SPLINE
SPL {X  -162.820, Y  +465.690, Z    +0.000, E1   -36.140, E3 +383343.973}
SPL {X  -162.820, Y  +470.432, Z    +0.000, E1   -36.100, E3 +383357.855}
SPL {X  -162.820, Y  +475.701, Z    +0.000, E1   -36.157, E3 +383372.483}
SPL {X  -162.820, Y  +479.954, Z    +0.000, E1   -36.086, E3 +383385.023}
SPL {X  -162.820, Y  +485.438, Z    +0.000, E1   -36.112, E3 +383400.741}
SPL {X  -162.820, Y  +490.843, Z    +0.000, E1   -36.087, E3 +383416.154}
SPL {X  -162.820, Y  +494.712, Z    +0.000, E1   -36.164, E3 +383426.667}
SPL {X  -162.820, Y  +497.796, Z    +0.000, E1   -36.022, E3 +383436.373}
SPL {X  -162.820, Y  +502.146, Z    +0.000, E1   -36.123, E3 +383448.242}
SPL {X  -162.820, Y  +505.688, Z    +0.000, E1   -36.050, E3 +383458.724}
SPL {X  -162.820, Y  +509.364, Z    +0.000, E1   -36.084, E3 +383469.095}
SPL {X  -162.820, Y  +513.393, Z    +0.000, E1   -36.179, E3 +383479.950}
SPL {X  -162.820, Y  +516.436, Z    +0.000, E1   -36.094, E3 +383489.146}
SPL {X  -162.820, Y  +520.482, Z    +0.000, E1   -36.096, E3 +383500.778}
SPL {X  -162.820, Y  +524.107, Z    +0.000, E1   -36.045, E3 +383511.362}
SPL {X  -162.820, Y  +527.962, Z    +0.000, E1   -36.074, E3 +383522.295}
SPL {X  -162.820, Y  +532.253, Z    +0.000, E1   -36.170, E3 +383533.884}
SPL {X  -162.820, Y  +536.031, Z    +0.000, E1   -36.058, E3 +383545.422}
SPL {X  -162.820, Y  +541.179, Z    +0.000, E1   -36.085, E3 +383560.062}
SPL {X  -162.820, Y  +546.355, Z    +0.000, E1   -36.114, E3 +383574.607}
SPL {X  -162.820, Y  +551.776, Z    +0.000, E1   -36.108, E3 +383590.240}
SPL {X  -162.820, Y  +558.272, Z    +0.000, E1   -36.170, E3 +383608.449}
SPL {X  -162.820, Y  +562.721, Z    +0.000, E1   -36.046, E3 +383621.674}
SPL {X  -162.820, Y  +566.500, Z    +0.000, E1   -36.073, E3 +383632.406}
SPL {X  -162.820, Y  +570.319, Z    +0.000, E1   -36.045, E3 +383643.434}
SPL {X  -162.820, Y  +573.265, Z    +0.000, E1   -36.071, E3 +383651.671}
SPL {X  -162.820, Y  +576.887, Z    +0.000, E1   -36.084, E3 +383662.029}
SPL {X  -162.820, Y  +581.763, Z    +0.000, E1   -36.093, E3 +383675.966}
SPL {X  -162.820, Y  +586.693, Z    +0.000, E1   -36.086, E3 +383690.071}
SPL {X  -162.820, Y  +591.665, Z    +0.000, E1   -36.045, E3 +383704.599}
SPL {X  -162.820, Y  +597.399, Z    +0.000, E1   -36.147, E3 +383720.362}
SPL {X  -162.820, Y  +602.243, Z    +0.000, E1   -36.085, E3 +383734.508}
SPL {X  -162.820, Y  +605.848, Z    +0.000, E1   -36.070, E3 +383744.829}
SPL {X  -162.820, Y  +609.375, Z    +0.000, E1   -36.084, E3 +383754.879}
SPL {X  -162.820, Y  +612.959, Z    +0.000, E1   -36.034, E3 +383765.400}
SPL {X  -162.820, Y  +616.897, Z    +0.000, E1   -36.061, E3 +383776.547}
SPL {X  -162.820, Y  +621.516, Z    +0.000, E1   -36.072, E3 +383789.746}
SPL {X  -162.820, Y  +626.243, Z    +0.000, E1   -36.105, E3 +383802.989}
SPL {X  -162.820, Y  +630.571, Z    +0.000, E1   -36.057, E3 +383815.691}
SPL {X  -162.820, Y  +634.189, Z    +0.000, E1   -36.065, E3 +383825.885}
SPL {X  -162.820, Y  +638.473, Z    +0.000, E1   -36.098, E3 +383838.122}
SPL {X  -162.820, Y  +642.832, Z    +0.000, E1   -36.091, E3 +383850.448}
SPL {X  -162.820, Y  +646.320, Z    +0.000, E1   -36.078, E3 +383860.555}
SPL {X  -162.820, Y  +649.997, Z    +0.000, E1   -36.000, E3 +383871.525}
SPL {X  -162.820, Y  +655.571, Z    +0.000, E1   -36.141, E3 +383886.860}
SPL {X  -162.820, Y  +661.560, Z    +0.000, E1   -36.068, E3 +383904.287}
SPL {X  -162.820, Y  +667.641, Z    +0.000, E1   -36.092, E3 +383921.668}
SPL {X  -162.820, Y  +673.415, Z    +0.000, E1   -36.053, E3 +383938.259}
SPL {X  -162.761, Y  +677.889, Z    +0.000, E1   -36.122, E3 +383950.577}
SPL {X  -162.577, Y  +682.401, Z    +0.000, E1   -36.021, E3 +383964.193}
SPL {X  -162.187, Y  +687.846, Z    +0.000, E1   -36.007, E3 +383979.862}
SPL {X  -161.667, Y  +692.839, Z    +0.000, E1   -35.918, E3 +383994.628}
SPL {X  -161.078, Y  +697.256, Z    +0.000, E1   -35.797, E3 +384007.964}
SPL {X  -160.313, Y  +701.964, Z    +0.000, E1   -35.709, E3 +384022.039}
SPL {X  -159.317, Y  +707.091, Z    +0.000, E1   -35.482, E3 +384038.063}
SPL {X  -158.510, Y  +710.714, Z    +0.000, E1   -35.230, E3 +384049.774}
SPL {X  -155.037, Y  +723.239, Z    +0.000, E1   -39.382, E3 +384058.870}
SPL {X  -152.141, Y  +731.494, Z    +0.000, E1   -35.181, E3 +384117.676}
ENDSPLINE

SPLINE
SPL {X  -152.670, Y  +730.088, Z    +0.000, E1   -30.916, E3 +384191.038}
SPL {X  -160.727, Y  +699.521, Z    +0.000, E1   -18.202, E3 +384157.321}
SPL {X  -161.979, Y  +690.023, Z    +0.000, E1   -12.991, E3 +384164.131}
SPL {X  -162.641, Y  +681.139, Z    +0.000, E1    -7.893, E3 +384166.223}
SPL {X  -162.820, Y  +673.062, Z    +0.000, E1    -2.992, E3 +384165.190}
SPL {X  -162.820, Y  +666.731, Z    +0.000, E1    +1.545, E3 +384166.820}
SPL {X  -162.820, Y  +660.758, Z    +0.000, E1    +6.523, E3 +384166.530}
SPL {X  -162.820, Y  +650.583, Z    +0.000, E1   +16.035, E3 +384165.503}
SPL {X  -162.820, Y  +629.267, Z    +0.000, E1   +31.872, E3 +384176.651}
SPL {X  -162.820, Y  +620.680, Z    +0.000, E1   +34.107, E3 +384190.701}
SPL {X  -162.820, Y  +601.185, Z    +0.000, E1   +39.430, E3 +384214.208}
SPL {X  -162.820, Y  +599.927, Z    +0.000, E1   +35.241, E3 +384240.786}
SPL {X  -162.820, Y  +599.021, Z    +0.000, E1   +33.912, E3 +384251.837}
SPL {X  -162.820, Y  +595.170, Z    +0.000, E1   +33.784, E3 +384264.743}
SPL {X  -162.820, Y  +589.785, Z    +0.000, E1   +33.904, E3 +384280.740}
SPL {X  -162.820, Y  +584.646, Z    +0.000, E1   +33.882, E3 +384296.809}
SPL {X  -162.820, Y  +579.919, Z    +0.000, E1   +33.857, E3 +384311.597}
SPL {X  -162.820, Y  +574.615, Z    +0.000, E1   +33.920, E3 +384327.771}
SPL {X  -162.820, Y  +569.298, Z    +0.000, E1   +33.851, E3 +384344.633}
SPL {X  -162.820, Y  +563.983, Z    +0.000, E1   +33.916, E3 +384360.774}
SPL {X  -162.820, Y  +559.395, Z    +0.000, E1   +33.796, E3 +384375.655}
SPL {X  -162.820, Y  +554.453, Z    +0.000, E1   +33.841, E3 +384390.880}
SPL {X  -162.820, Y  +548.576, Z    +0.000, E1   +33.950, E3 +384408.410}
SPL {X  -162.820, Y  +544.808, Z    +0.000, E1   +33.827, E3 +384420.673}
SPL {X  -162.820, Y  +541.668, Z    +0.000, E1   +33.787, E3 +384430.779}
SPL {X  -162.820, Y  +537.061, Z    +0.000, E1   +33.897, E3 +384444.437}
SPL {X  -162.820, Y  +532.164, Z    +0.000, E1   +33.861, E3 +384459.911}
SPL {X  -162.820, Y  +526.783, Z    +0.000, E1   +33.870, E3 +384476.594}
SPL {X  -162.820, Y  +521.520, Z    +0.000, E1   +33.826, E3 +384493.241}
SPL {X  -162.820, Y  +515.754, Z    +0.000, E1   +33.911, E3 +384510.643}
SPL {X  -162.820, Y  +510.207, Z    +0.000, E1   +33.879, E3 +384528.023}
SPL {X  -162.820, Y  +505.651, Z    +0.000, E1   +33.839, E3 +384542.317}
SPL {X  -162.820, Y  +500.931, Z    +0.000, E1   +34.256, E3 +384554.190}
SPL {X  -162.820, Y  +481.122, Z    +0.000, E1   +41.279, E3 +384564.455}
SPL {X  -162.820, Y  +478.698, Z    +0.000, E1   +40.526, E3 +384574.804}
SPL {X  -162.820, Y  +475.203, Z    +0.000, E1   +39.596, E3 +384589.263}
SPL {X  -162.820, Y  +472.097, Z    +0.000, E1   +38.411, E3 +384604.230}
SPL {X  -162.820, Y  +469.308, Z    +0.000, E1   +37.839, E3 +384615.034}
SPL {X  -162.820, Y  +467.216, Z    +0.000, E1   +37.215, E3 +384624.601}
SPL {X  -162.820, Y  +462.598, Z    +0.000, E1   +37.325, E3 +384636.555}
SPL {X  -162.820, Y  +457.832, Z    +0.000, E1   +37.294, E3 +384649.841}
SPL {X  -162.820, Y  +452.986, Z    +0.000, E1   +37.368, E3 +384662.575}
SPL {X  -162.820, Y  +447.084, Z    +0.000, E1   +37.389, E3 +384678.766}
SPL {X  -162.820, Y  +440.036, Z    +0.000, E1   +37.326, E3 +384698.384}
SPL {X  -162.820, Y  +434.320, Z    +0.000, E1   +37.343, E3 +384713.707}
SPL {X  -162.820, Y  +430.091, Z    +0.000, E1   +37.424, E3 +384724.707}
SPL {X  -162.820, Y  +426.177, Z    +0.000, E1   +37.250, E3 +384736.530}
SPL {X  -162.820, Y  +421.391, Z    +0.000, E1   +37.346, E3 +384748.994}
SPL {X  -162.820, Y  +416.811, Z    +0.000, E1   +37.348, E3 +384761.528}
SPL {X  -162.820, Y  +411.860, Z    +0.000, E1   +37.402, E3 +384774.680}
SPL {X  -162.820, Y  +407.726, Z    +0.000, E1   +37.291, E3 +384786.627}
SPL {X  -162.820, Y  +403.543, Z    +0.000, E1   +37.305, E3 +384797.973}
SPL {X  -162.820, Y  +399.300, Z    +0.000, E1   +37.355, E3 +384809.257}
SPL {X  -162.820, Y  +395.182, Z    +0.000, E1   +37.347, E3 +384820.546}
SPL {X  -162.820, Y  +390.797, Z    +0.000, E1   +37.358, E3 +384832.458}
SPL {X  -162.820, Y  +386.671, Z    +0.000, E1   +37.363, E3 +384843.639}
SPL {X  -162.820, Y  +382.174, Z    +0.000, E1   +37.329, E3 +384856.217}
SPL {X  -162.785, Y  +377.133, Z    +0.000, E1   +37.299, E3 +384870.146}
SPL {X  -162.623, Y  +372.484, Z    +0.000, E1   +37.337, E3 +384882.586}
SPL {X  -162.331, Y  +367.894, Z    +0.000, E1   +37.251, E3 +384895.698}
SPL {X  -161.920, Y  +363.407, Z    +0.000, E1   +37.164, E3 +384908.432}
SPL {X  -161.482, Y  +359.669, Z    +0.000, E1   +37.064, E3 +384919.217}
SPL {X  -160.943, Y  +355.851, Z    +0.000, E1   +37.136, E3 +384929.203}
SPL {X  -160.493, Y  +353.069, Z    +0.000, E1   +36.789, E3 +384938.855}
SPL {X  -159.837, Y  +349.474, Z    +0.000, E1   +36.824, E3 +384948.521}
SPL {X  -158.862, Y  +344.820, Z    +0.000, E1   +36.732, E3 +384961.884}
SPL {X  -157.959, Y  +341.011, Z    +0.000, E1   +36.448, E3 +384973.780}
SPL {X  -153.520, Y  +326.260, Z    +0.000, E1   +41.363, E3 +384982.613}
SPL {X  -150.942, Y  +319.452, Z    +0.000, E1   +36.529, E3 +385038.970}
ENDSPLINE

SPLINE
SPL {X  -159.264, Y  +346.659, Z    +0.000, E1   +22.083, E3 +385079.544}
SPL {X  -161.245, Y  +357.907, Z    +0.000, E1   +16.095, E3 +385092.977}
SPL {X  -162.697, Y  +374.161, Z    +0.000, E1    +7.119, E3 +385090.966}
SPL {X  -162.820, Y  +380.878, Z    +0.000, E1    +2.854, E3 +385093.797}
SPL {X  -162.820, Y  +385.313, Z    +0.000, E1    -0.228, E3 +385093.578}
SPL {X  -162.820, Y  +389.965, Z    +0.000, E1    -3.918, E3 +385092.946}
SPL {X  -162.820, Y  +394.532, Z    +0.000, E1    -7.849, E3 +385094.494}
SPL {X  -162.820, Y  +400.765, Z    +0.000, E1   -14.108, E3 +385091.961}
SPL {X  -162.820, Y  +411.829, Z    +0.000, E1   -24.195, E3 +385094.039}
SPL {X  -162.820, Y  +434.900, Z    +0.000, E1   -34.666, E3 +385121.403}
SPL {X  -162.820, Y  +465.031, Z    +0.000, E1   -41.710, E3 +385159.076}
SPL {X  -162.820, Y  +465.893, Z    +0.000, E1   -40.572, E3 +385167.605}
ENDSPLINE

SPLINE
SPL {X  -162.820, Y  +458.794, Z    +0.000, E1   -36.100, E3 +385176.334}
ENDSPLINE

SPLINE
SPL {X  -162.820, Y  +461.779, Z    +0.000, E1   -35.988, E3 +385185.530}
SPL {X  -162.820, Y  +465.690, Z    +0.000, E1   -36.140, E3 +385195.825}
SPL {X  -162.820, Y  +470.432, Z    +0.000, E1   -36.100, E3 +385209.707}
SPL {X  -162.820, Y  +475.701, Z    +0.000, E1   -36.157, E3 +385224.334}
SPL {X  -162.820, Y  +479.954, Z    +0.000, E1   -36.086, E3 +385236.875}
SPL {X  -162.820, Y  +483.976, Z    +0.000, E1   -36.049, E3 +385248.607}
SPL {X  -162.820, Y  +488.601, Z    +0.000, E1   -36.081, E3 +385261.697}
SPL {X  -162.820, Y  +493.837, Z    +0.000, E1   -36.178, E3 +385276.040}
SPL {X  -162.820, Y  +498.932, Z    +0.000, E1   -36.079, E3 +385291.245}
SPL {X  -162.820, Y  +504.528, Z    +0.000, E1   -36.109, E3 +385307.041}
SPL {X  -162.820, Y  +509.364, Z    +0.000, E1   -36.084, E3 +385320.946}
SPL {X  -162.820, Y  +515.001, Z    +0.000, E1   -36.183, E3 +385336.584}
SPL {X  -162.820, Y  +520.482, Z    +0.000, E1   -36.096, E3 +385352.630}
SPL {X  -162.820, Y  +524.107, Z    +0.000, E1   -36.045, E3 +385363.214}
SPL {X  -162.820, Y  +527.962, Z    +0.000, E1   -36.074, E3 +385374.146}
SPL {X  -162.820, Y  +532.253, Z    +0.000, E1   -36.170, E3 +385385.735}
SPL {X  -162.820, Y  +536.031, Z    +0.000, E1   -36.058, E3 +385397.273}
SPL {X  -162.820, Y  +541.179, Z    +0.000, E1   -36.085, E3 +385411.914}
SPL {X  -162.820, Y  +546.355, Z    +0.000, E1   -36.114, E3 +385426.458}
SPL {X  -162.820, Y  +551.776, Z    +0.000, E1   -36.108, E3 +385442.092}
SPL {X  -162.820, Y  +556.944, Z    +0.000, E1   -36.118, E3 +385456.663}
SPL {X  -162.820, Y  +561.684, Z    +0.000, E1   -36.118, E3 +385470.255}
SPL {X  -162.820, Y  +566.500, Z    +0.000, E1   -36.073, E3 +385484.258}
SPL {X  -162.820, Y  +571.734, Z    +0.000, E1   -36.094, E3 +385499.187}
SPL {X  -162.820, Y  +576.887, Z    +0.000, E1   -36.084, E3 +385513.881}
SPL {X  -162.820, Y  +581.763, Z    +0.000, E1   -36.093, E3 +385527.818}
SPL {X  -162.820, Y  +586.693, Z    +0.000, E1   -36.086, E3 +385541.923}
SPL {X  -162.820, Y  +591.665, Z    +0.000, E1   -36.045, E3 +385556.450}
SPL {X  -162.820, Y  +597.399, Z    +0.000, E1   -36.147, E3 +385572.214}
SPL {X  -162.820, Y  +602.243, Z    +0.000, E1   -36.085, E3 +385586.360}
SPL {X  -162.820, Y  +606.975, Z    +0.000, E1   -36.102, E3 +385599.805}
SPL {X  -162.820, Y  +611.980, Z    +0.000, E1   -36.072, E3 +385614.351}
SPL {X  -162.820, Y  +616.897, Z    +0.000, E1   -36.061, E3 +385628.399}
SPL {X  -162.820, Y  +621.516, Z    +0.000, E1   -36.072, E3 +385641.598}
SPL {X  -162.820, Y  +626.243, Z    +0.000, E1   -36.105, E3 +385654.841}
SPL {X  -162.820, Y  +630.571, Z    +0.000, E1   -36.057, E3 +385667.543}
SPL {X  -162.820, Y  +635.505, Z    +0.000, E1   -36.079, E3 +385681.549}
SPL {X  -162.820, Y  +641.277, Z    +0.000, E1   -36.126, E3 +385697.841}
SPL {X  -162.820, Y  +646.320, Z    +0.000, E1   -36.078, E3 +385712.407}
SPL {X  -162.820, Y  +651.289, Z    +0.000, E1   -36.059, E3 +385726.863}
SPL {X  -162.820, Y  +656.677, Z    +0.000, E1   -36.110, E3 +385741.876}
SPL {X  -162.820, Y  +661.560, Z    +0.000, E1   -36.068, E3 +385756.139}
SPL {X  -162.820, Y  +667.641, Z    +0.000, E1   -36.092, E3 +385773.520}
SPL {X  -162.820, Y  +673.415, Z    +0.000, E1   -36.053, E3 +385790.111}
SPL {X  -162.761, Y  +677.889, Z    +0.000, E1   -36.122, E3 +385802.429}
SPL {X  -162.577, Y  +682.401, Z    +0.000, E1   -36.021, E3 +385816.045}
SPL {X  -162.296, Y  +686.558, Z    +0.000, E1   -35.952, E3 +385828.236}
SPL {X  -161.948, Y  +690.331, Z    +0.000, E1   -35.960, E3 +385839.034}
SPL {X  -161.544, Y  +693.846, Z    +0.000, E1   -35.908, E3 +385849.309}
SPL {X  -160.925, Y  +698.267, Z    +0.000, E1   -35.816, E3 +385862.741}
SPL {X  -160.151, Y  +702.861, Z    +0.000, E1   -35.643, E3 +385876.711}
SPL {X  -159.317, Y  +707.091, Z    +0.000, E1   -35.482, E3 +385889.915}
SPL {X  -158.510, Y  +710.714, Z    +0.000, E1   -35.230, E3 +385901.626}
SPL {X  -155.037, Y  +723.239, Z    +0.000, E1   -39.382, E3 +385910.722}
SPL {X  -152.141, Y  +731.494, Z    +0.000, E1   -35.181, E3 +385969.528}
ENDSPLINE

SPLINE
SPL {X  -152.670, Y  +730.088, Z    +0.000, E1   -30.916, E3 +386042.890}
SPL {X  -160.727, Y  +699.521, Z    +0.000, E1   -18.202, E3 +386009.173}
SPL {X  -161.979, Y  +690.023, Z    +0.000, E1   -12.991, E3 +386015.983}
SPL {X  -162.641, Y  +681.139, Z    +0.000, E1    -7.893, E3 +386018.075}
SPL {X  -162.815, Y  +674.833, Z    +0.000, E1    -4.093, E3 +386015.690}
SPL {X  -162.820, Y  +669.862, Z    +0.000, E1    -0.751, E3 +386018.909}
SPL {X  -162.820, Y  +664.572, Z    +0.000, E1    +3.252, E3 +386018.722}
SPL {X  -162.820, Y  +657.781, Z    +0.000, E1    +9.391, E3 +386016.545}
SPL {X  -162.820, Y  +648.706, Z    +0.000, E1   +17.761, E3 +386018.297}
SPL {X  -162.820, Y  +635.926, Z    +0.000, E1   +28.192, E3 +386023.124}
SPL {X  -162.820, Y  +621.673, Z    +0.000, E1   +34.265, E3 +386039.482}
SPL {X  -162.820, Y  +609.002, Z    +0.000, E1   +38.458, E3 +386052.704}
SPL {X  -162.820, Y  +596.392, Z    +0.000, E1   +37.895, E3 +386086.173}
ENDSPLINE

SPLINE
SPL {X  -162.820, Y  +601.432, Z    +0.000, E1   +34.026, E3 +386095.470}
ENDSPLINE

SPLINE
SPL {X  -162.820, Y  +597.570, Z    +0.000, E1   +33.919, E3 +386108.368}
SPL {X  -162.820, Y  +592.692, Z    +0.000, E1   +33.779, E3 +386124.260}
SPL {X  -162.820, Y  +588.795, Z    +0.000, E1   +33.876, E3 +386135.697}
SPL {X  -162.820, Y  +584.646, Z    +0.000, E1   +33.882, E3 +386148.661}
SPL {X  -162.820, Y  +579.919, Z    +0.000, E1   +33.857, E3 +386163.449}
SPL {X  -162.820, Y  +576.636, Z    +0.000, E1   +33.845, E3 +386173.595}
SPL {X  -162.820, Y  +573.566, Z    +0.000, E1   +33.899, E3 +386182.844}
SPL {X  -162.820, Y  +570.335, Z    +0.000, E1   +33.821, E3 +386193.328}
SPL {X  -162.820, Y  +565.901, Z    +0.000, E1   +33.889, E3 +386206.849}
SPL {X  -162.820, Y  +562.173, Z    +0.000, E1   +33.897, E3 +386218.140}
SPL {X  -162.820, Y  +558.179, Z    +0.000, E1   +33.857, E3 +386231.075}
SPL {X  -162.820, Y  +553.486, Z    +0.000, E1   +33.777, E3 +386245.980}
SPL {X  -162.820, Y  +549.726, Z    +0.000, E1   +33.905, E3 +386256.835}
SPL {X  -162.820, Y  +545.760, Z    +0.000, E1   +33.901, E3 +386269.231}
SPL {X  -162.820, Y  +541.668, Z    +0.000, E1   +33.787, E3 +386282.631}
SPL {X  -162.820, Y  +538.174, Z    +0.000, E1   +33.865, E3 +386292.920}
SPL {X  -162.820, Y  +534.943, Z    +0.000, E1   +33.919, E3 +386302.661}
SPL {X  -162.820, Y  +531.459, Z    +0.000, E1   +33.783, E3 +386314.318}
SPL {X  -162.820, Y  +526.783, Z    +0.000, E1   +33.870, E3 +386328.446}
SPL {X  -162.820, Y  +521.520, Z    +0.000, E1   +33.826, E3 +386345.093}
SPL {X  -162.820, Y  +516.814, Z    +0.000, E1   +33.917, E3 +386358.994}
SPL {X  -162.820, Y  +512.685, Z    +0.000, E1   +33.830, E3 +386372.437}
SPL {X  -162.820, Y  +508.888, Z    +0.000, E1   +33.871, E3 +386383.852}
SPL {X  -162.820, Y  +505.651, Z    +0.000, E1   +33.839, E3 +386394.169}
SPL {X  -162.820, Y  +500.931, Z    +0.000, E1   +34.256, E3 +386406.042}
SPL {X  -162.820, Y  +481.122, Z    +0.000, E1   +41.279, E3 +386416.307}
SPL {X  -162.820, Y  +478.698, Z    +0.000, E1   +40.526, E3 +386426.656}
SPL {X  -162.820, Y  +475.203, Z    +0.000, E1   +39.596, E3 +386441.115}
SPL {X  -162.820, Y  +472.097, Z    +0.000, E1   +38.411, E3 +386456.082}
SPL {X  -162.820, Y  +469.308, Z    +0.000, E1   +37.839, E3 +386466.886}
SPL {X  -162.820, Y  +467.216, Z    +0.000, E1   +37.215, E3 +386476.452}
SPL {X  -162.820, Y  +462.598, Z    +0.000, E1   +37.325, E3 +386488.407}
SPL {X  -162.820, Y  +459.177, Z    +0.000, E1   +37.207, E3 +386498.434}
SPL {X  -162.820, Y  +453.939, Z    +0.000, E1   +37.397, E3 +386511.786}
SPL {X  -162.820, Y  +447.084, Z    +0.000, E1   +37.389, E3 +386530.618}
SPL {X  -162.820, Y  +440.036, Z    +0.000, E1   +37.326, E3 +386550.235}
SPL {X  -162.820, Y  +434.320, Z    +0.000, E1   +37.343, E3 +386565.559}
SPL {X  -162.820, Y  +430.091, Z    +0.000, E1   +37.424, E3 +386576.559}
SPL {X  -162.820, Y  +426.177, Z    +0.000, E1   +37.250, E3 +386588.382}
SPL {X  -162.820, Y  +421.391, Z    +0.000, E1   +37.346, E3 +386600.845}
SPL {X  -162.820, Y  +416.811, Z    +0.000, E1   +37.348, E3 +386613.380}
SPL {X  -162.820, Y  +411.860, Z    +0.000, E1   +37.402, E3 +386626.531}
SPL {X  -162.820, Y  +407.726, Z    +0.000, E1   +37.291, E3 +386638.479}
SPL {X  -162.820, Y  +403.543, Z    +0.000, E1   +37.305, E3 +386649.825}
SPL {X  -162.820, Y  +399.300, Z    +0.000, E1   +37.355, E3 +386661.109}
SPL {X  -162.820, Y  +395.182, Z    +0.000, E1   +37.347, E3 +386672.398}
SPL {X  -162.820, Y  +390.797, Z    +0.000, E1   +37.358, E3 +386684.310}
SPL {X  -162.820, Y  +386.671, Z    +0.000, E1   +37.363, E3 +386695.491}
SPL {X  -162.820, Y  +382.174, Z    +0.000, E1   +37.329, E3 +386708.069}
SPL {X  -162.785, Y  +377.133, Z    +0.000, E1   +37.299, E3 +386721.998}
SPL {X  -162.576, Y  +371.586, Z    +0.000, E1   +37.322, E3 +386737.110}
SPL {X  -162.256, Y  +366.963, Z    +0.000, E1   +37.251, E3 +386749.999}
SPL {X  -161.920, Y  +363.407, Z    +0.000, E1   +37.164, E3 +386760.284}
SPL {X  -161.341, Y  +358.603, Z    +0.000, E1   +37.117, E3 +386773.764}
SPL {X  -160.616, Y  +353.801, Z    +0.000, E1   +36.942, E3 +386787.929}
SPL {X  -159.837, Y  +349.474, Z    +0.000, E1   +36.824, E3 +386800.373}
SPL {X  -158.862, Y  +344.820, Z    +0.000, E1   +36.732, E3 +386813.735}
SPL {X  -157.959, Y  +341.011, Z    +0.000, E1   +36.448, E3 +386825.632}
SPL {X  -153.520, Y  +326.260, Z    +0.000, E1   +41.363, E3 +386834.465}
SPL {X  -150.942, Y  +319.452, Z    +0.000, E1   +36.529, E3 +386890.821}
ENDSPLINE

SPLINE
SPL {X  -159.264, Y  +346.659, Z    +0.000, E1   +22.083, E3 +386931.396}
SPL {X  -161.245, Y  +357.907, Z    +0.000, E1   +16.095, E3 +386944.828}
SPL {X  -162.697, Y  +374.161, Z    +0.000, E1    +7.119, E3 +386942.818}
SPL {X  -162.820, Y  +380.878, Z    +0.000, E1    +2.854, E3 +386945.649}
SPL {X  -162.820, Y  +385.313, Z    +0.000, E1    -0.228, E3 +386945.429}
SPL {X  -162.820, Y  +389.965, Z    +0.000, E1    -3.918, E3 +386944.798}
SPL {X  -162.820, Y  +394.532, Z    +0.000, E1    -7.849, E3 +386946.346}
SPL {X  -162.820, Y  +400.765, Z    +0.000, E1   -14.108, E3 +386943.813}
SPL {X  -162.820, Y  +411.829, Z    +0.000, E1   -24.195, E3 +386945.890}
SPL {X  -162.820, Y  +434.900, Z    +0.000, E1   -34.666, E3 +386973.255}
SPL {X  -162.820, Y  +465.440, Z    +0.000, E1   -41.264, E3 +387014.562}
ENDSPLINE

SPLINE
SPL {X  -162.820, Y  +458.794, Z    +0.000, E1   -36.100, E3 +387028.186}
ENDSPLINE

SPLINE
SPL {X  -162.820, Y  +461.779, Z    +0.000, E1   -35.988, E3 +387037.382}
SPL {X  -162.820, Y  +465.690, Z    +0.000, E1   -36.140, E3 +387047.676}
SPL {X  -162.820, Y  +470.432, Z    +0.000, E1   -36.100, E3 +387061.559}
SPL {X  -162.820, Y  +475.701, Z    +0.000, E1   -36.157, E3 +387076.186}
SPL {X  -162.820, Y  +479.954, Z    +0.000, E1   -36.086, E3 +387088.727}
SPL {X  -162.820, Y  +483.976, Z    +0.000, E1   -36.049, E3 +387100.459}
SPL {X  -162.820, Y  +489.628, Z    +0.000, E1   -36.135, E3 +387116.289}
SPL {X  -162.820, Y  +494.712, Z    +0.000, E1   -36.164, E3 +387130.370}
SPL {X  -162.820, Y  +498.932, Z    +0.000, E1   -36.079, E3 +387143.097}
SPL {X  -162.820, Y  +504.528, Z    +0.000, E1   -36.109, E3 +387158.893}
SPL {X  -162.820, Y  +509.364, Z    +0.000, E1   -36.084, E3 +387172.798}
SPL {X  -162.820, Y  +515.001, Z    +0.000, E1   -36.183, E3 +387188.436}
SPL {X  -162.820, Y  +520.482, Z    +0.000, E1   -36.096, E3 +387204.482}
SPL {X  -162.820, Y  +525.226, Z    +0.000, E1   -36.081, E3 +387218.149}
SPL {X  -162.820, Y  +530.908, Z    +0.000, E1   -36.155, E3 +387234.007}
SPL {X  -162.820, Y  +536.031, Z    +0.000, E1   -36.058, E3 +387249.125}
SPL {X  -162.820, Y  +541.179, Z    +0.000, E1   -36.085, E3 +387263.766}
SPL {X  -162.820, Y  +546.355, Z    +0.000, E1   -36.114, E3 +387278.310}
SPL {X  -162.820, Y  +551.776, Z    +0.000, E1   -36.108, E3 +387293.944}
SPL {X  -162.820, Y  +556.944, Z    +0.000, E1   -36.118, E3 +387308.515}
SPL {X  -162.820, Y  +561.684, Z    +0.000, E1   -36.118, E3 +387322.107}
SPL {X  -162.820, Y  +566.500, Z    +0.000, E1   -36.073, E3 +387336.110}
SPL {X  -162.820, Y  +571.734, Z    +0.000, E1   -36.094, E3 +387351.039}
SPL {X  -162.820, Y  +576.887, Z    +0.000, E1   -36.084, E3 +387365.733}
SPL {X  -162.820, Y  +581.763, Z    +0.000, E1   -36.093, E3 +387379.670}
SPL {X  -162.820, Y  +586.693, Z    +0.000, E1   -36.086, E3 +387393.774}
SPL {X  -162.820, Y  +590.250, Z    +0.000, E1   -36.075, E3 +387403.893}
SPL {X  -162.820, Y  +592.727, Z    +0.000, E1   -35.960, E3 +387411.717}
SPL {X  -162.820, Y  +597.399, Z    +0.000, E1   -36.147, E3 +387424.066}
SPL {X  -162.820, Y  +602.243, Z    +0.000, E1   -36.085, E3 +387438.212}
SPL {X  -162.820, Y  +606.975, Z    +0.000, E1   -36.102, E3 +387451.657}
SPL {X  -162.820, Y  +611.980, Z    +0.000, E1   -36.072, E3 +387466.202}
SPL {X  -162.820, Y  +616.897, Z    +0.000, E1   -36.061, E3 +387480.251}
SPL {X  -162.820, Y  +621.516, Z    +0.000, E1   -36.072, E3 +387493.450}
SPL {X  -162.820, Y  +626.243, Z    +0.000, E1   -36.105, E3 +387506.693}
SPL {X  -162.820, Y  +630.571, Z    +0.000, E1   -36.057, E3 +387519.395}
SPL {X  -162.820, Y  +634.189, Z    +0.000, E1   -36.065, E3 +387529.588}
SPL {X  -162.820, Y  +638.473, Z    +0.000, E1   -36.098, E3 +387541.825}
SPL {X  -162.820, Y  +642.832, Z    +0.000, E1   -36.091, E3 +387554.151}
SPL {X  -162.820, Y  +646.320, Z    +0.000, E1   -36.078, E3 +387564.258}
SPL {X  -162.820, Y  +651.289, Z    +0.000, E1   -36.059, E3 +387578.715}
SPL {X  -162.820, Y  +656.677, Z    +0.000, E1   -36.110, E3 +387593.728}
SPL {X  -162.820, Y  +661.560, Z    +0.000, E1   -36.068, E3 +387607.991}
SPL {X  -162.820, Y  +666.386, Z    +0.000, E1   -36.048, E3 +387621.875}
SPL {X  -162.820, Y  +671.104, Z    +0.000, E1   -36.061, E3 +387635.295}
SPL {X  -162.787, Y  +676.764, Z    +0.000, E1   -36.126, E3 +387651.194}
SPL {X  -162.633, Y  +681.311, Z    +0.000, E1   -35.984, E3 +387664.883}
SPL {X  -162.367, Y  +685.641, Z    +0.000, E1   -36.000, E3 +387677.291}
SPL {X  -162.041, Y  +689.412, Z    +0.000, E1   -36.001, E3 +387687.910}
SPL {X  -161.667, Y  +692.839, Z    +0.000, E1   -35.918, E3 +387698.331}
SPL {X  -161.078, Y  +697.256, Z    +0.000, E1   -35.797, E3 +387711.668}
SPL {X  -160.313, Y  +701.964, Z    +0.000, E1   -35.709, E3 +387725.743}
SPL {X  -159.622, Y  +705.613, Z    +0.000, E1   -35.430, E3 +387737.682}
SPL {X  -158.758, Y  +709.640, Z    +0.000, E1   -35.380, E3 +387749.689}
SPL {X  -155.037, Y  +723.239, Z    +0.000, E1   -39.382, E3 +387762.574}
SPL {X  -152.141, Y  +731.494, Z    +0.000, E1   -35.181, E3 +387821.380}
ENDSPLINE

SPLINE
SPL {X  -160.133, Y  +702.956, Z    +0.000, E1   -19.806, E3 +387864.918}
SPL {X  -161.979, Y  +690.023, Z    +0.000, E1   -12.991, E3 +387867.835}
SPL {X  -162.783, Y  +676.950, Z    +0.000, E1    -5.489, E3 +387868.365}
SPL {X  -162.820, Y  +669.862, Z    +0.000, E1    -0.751, E3 +387870.760}
SPL {X  -162.820, Y  +665.790, Z    +0.000, E1    +2.338, E3 +387870.133}
SPL {X  -162.820, Y  +660.758, Z    +0.000, E1    +6.523, E3 +387870.234}
SPL {X  -162.820, Y  +650.583, Z    +0.000, E1   +16.035, E3 +387869.206}
SPL {X  -162.820, Y  +629.267, Z    +0.000, E1   +31.872, E3 +387880.355}
SPL {X  -162.820, Y  +620.680, Z    +0.000, E1   +34.107, E3 +387894.404}
SPL {X  -162.820, Y  +609.002, Z    +0.000, E1   +38.458, E3 +387904.556}
SPL {X  -162.820, Y  +596.392, Z    +0.000, E1   +37.895, E3 +387938.024}
ENDSPLINE

SPLINE
SPL {X  -162.820, Y  +599.924, Z    +0.000, E1   +33.992, E3 +387952.398}
ENDSPLINE

SPLINE
SPL {X  -162.820, Y  +596.128, Z    +0.000, E1   +33.827, E3 +387965.036}
SPL {X  -162.820, Y  +592.692, Z    +0.000, E1   +33.779, E3 +387976.112}
SPL {X  -162.820, Y  +588.795, Z    +0.000, E1   +33.876, E3 +387987.548}
SPL {X  -162.820, Y  +585.519, Z    +0.000, E1   +33.888, E3 +387997.633}
SPL {X  -162.820, Y  +582.066, Z    +0.000, E1   +33.857, E3 +388008.567}
SPL {X  -162.820, Y  +577.919, Z    +0.000, E1   +33.841, E3 +388021.621}
SPL {X  -162.820, Y  +573.566, Z    +0.000, E1   +33.899, E3 +388034.695}
SPL {X  -162.820, Y  +569.298, Z    +0.000, E1   +33.851, E3 +388048.337}
SPL {X  -162.820, Y  +565.024, Z    +0.000, E1   +33.872, E3 +388061.393}
SPL {X  -162.820, Y  +560.226, Z    +0.000, E1   +33.868, E3 +388076.486}
SPL {X  -162.820, Y  +554.453, Z    +0.000, E1   +33.841, E3 +388094.583}
SPL {X  -162.820, Y  +548.576, Z    +0.000, E1   +33.950, E3 +388112.114}
SPL {X  -162.820, Y  +544.808, Z    +0.000, E1   +33.827, E3 +388124.377}
SPL {X  -162.820, Y  +541.668, Z    +0.000, E1   +33.787, E3 +388134.483}
SPL {X  -162.820, Y  +538.174, Z    +0.000, E1   +33.865, E3 +388144.772}
SPL {X  -162.820, Y  +534.943, Z    +0.000, E1   +33.919, E3 +388154.512}
SPL {X  -162.820, Y  +530.273, Z    +0.000, E1   +33.855, E3 +388169.542}
SPL {X  -162.820, Y  +524.900, Z    +0.000, E1   +33.820, E3 +388186.442}
SPL {X  -162.820, Y  +520.532, Z    +0.000, E1   +33.805, E3 +388200.010}
SPL {X  -162.820, Y  +516.814, Z    +0.000, E1   +33.917, E3 +388210.846}
SPL {X  -162.820, Y  +512.685, Z    +0.000, E1   +33.830, E3 +388224.289}
SPL {X  -162.820, Y  +508.888, Z    +0.000, E1   +33.871, E3 +388235.704}
SPL {X  -162.820, Y  +505.651, Z    +0.000, E1   +33.839, E3 +388246.021}
SPL {X  -162.820, Y  +500.931, Z    +0.000, E1   +34.256, E3 +388257.894}
SPL {X  -162.820, Y  +481.122, Z    +0.000, E1   +41.279, E3 +388268.158}
SPL {X  -162.820, Y  +478.698, Z    +0.000, E1   +40.526, E3 +388278.507}
SPL {X  -162.820, Y  +475.203, Z    +0.000, E1   +39.596, E3 +388292.967}
SPL {X  -162.820, Y  +472.097, Z    +0.000, E1   +38.411, E3 +388307.934}
SPL {X  -162.820, Y  +469.308, Z    +0.000, E1   +37.839, E3 +388318.738}
SPL {X  -162.820, Y  +467.216, Z    +0.000, E1   +37.215, E3 +388328.304}
SPL {X  -162.820, Y  +462.598, Z    +0.000, E1   +37.325, E3 +388340.258}
SPL {X  -162.820, Y  +457.832, Z    +0.000, E1   +37.294, E3 +388353.545}
SPL {X  -162.820, Y  +452.986, Z    +0.000, E1   +37.368, E3 +388366.279}
SPL {X  -162.820, Y  +448.311, Z    +0.000, E1   +37.333, E3 +388379.299}
SPL {X  -162.820, Y  +443.351, Z    +0.000, E1   +37.335, E3 +388392.829}
SPL {X  -162.820, Y  +438.727, Z    +0.000, E1   +37.289, E3 +388405.701}
SPL {X  -162.820, Y  +434.320, Z    +0.000, E1   +37.343, E3 +388417.411}
SPL {X  -162.820, Y  +430.091, Z    +0.000, E1   +37.424, E3 +388428.411}
SPL {X  -162.820, Y  +426.177, Z    +0.000, E1   +37.250, E3 +388440.234}
SPL {X  -162.820, Y  +421.391, Z    +0.000, E1   +37.346, E3 +388452.697}
SPL {X  -162.820, Y  +416.811, Z    +0.000, E1   +37.348, E3 +388465.232}
SPL {X  -162.820, Y  +411.860, Z    +0.000, E1   +37.402, E3 +388478.383}
SPL {X  -162.820, Y  +407.726, Z    +0.000, E1   +37.291, E3 +388490.331}
SPL {X  -162.820, Y  +403.543, Z    +0.000, E1   +37.305, E3 +388501.677}
SPL {X  -162.820, Y  +399.300, Z    +0.000, E1   +37.355, E3 +388512.961}
SPL {X  -162.820, Y  +395.182, Z    +0.000, E1   +37.347, E3 +388524.250}
SPL {X  -162.820, Y  +390.797, Z    +0.000, E1   +37.358, E3 +388536.162}
SPL {X  -162.820, Y  +386.671, Z    +0.000, E1   +37.363, E3 +388547.343}
SPL {X  -162.820, Y  +382.174, Z    +0.000, E1   +37.329, E3 +388559.920}
SPL {X  -162.785, Y  +377.133, Z    +0.000, E1   +37.299, E3 +388573.850}
SPL {X  -162.623, Y  +372.484, Z    +0.000, E1   +37.337, E3 +388586.289}
SPL {X  -162.331, Y  +367.894, Z    +0.000, E1   +37.251, E3 +388599.402}
SPL {X  -161.920, Y  +363.407, Z    +0.000, E1   +37.164, E3 +388612.136}
SPL {X  -161.341, Y  +358.603, Z    +0.000, E1   +37.117, E3 +388625.616}
SPL {X  -160.616, Y  +353.801, Z    +0.000, E1   +36.942, E3 +388639.781}
SPL {X  -159.837, Y  +349.474, Z    +0.000, E1   +36.824, E3 +388652.225}
SPL {X  -158.862, Y  +344.820, Z    +0.000, E1   +36.732, E3 +388665.587}
SPL {X  -157.959, Y  +341.011, Z    +0.000, E1   +36.448, E3 +388677.484}
SPL {X  -153.520, Y  +326.260, Z    +0.000, E1   +41.363, E3 +388686.316}
SPL {X  -150.942, Y  +319.452, Z    +0.000, E1   +36.529, E3 +388742.673}
ENDSPLINE

SPLINE
SPL {X  -159.264, Y  +346.659, Z    +0.000, E1   +22.083, E3 +388783.248}
SPL {X  -161.245, Y  +357.907, Z    +0.000, E1   +16.095, E3 +388796.680}
SPL {X  -162.746, Y  +375.590, Z    +0.000, E1    +6.280, E3 +388796.269}
SPL {X  -162.820, Y  +384.478, Z    +0.000, E1    +0.434, E3 +388796.938}
SPL {X  -162.820, Y  +389.965, Z    +0.000, E1    -3.918, E3 +388796.650}
SPL {X  -162.820, Y  +394.532, Z    +0.000, E1    -7.849, E3 +388798.198}
SPL {X  -162.820, Y  +400.765, Z    +0.000, E1   -14.108, E3 +388795.665}
SPL {X  -162.820, Y  +411.829, Z    +0.000, E1   -24.195, E3 +388797.742}
SPL {X  -162.820, Y  +434.900, Z    +0.000, E1   -34.666, E3 +388825.107}
SPL {X  -162.820, Y  +465.440, Z    +0.000, E1   -41.264, E3 +388866.414}
ENDSPLINE

SPLINE
SPL {X  -162.820, Y  +460.175, Z    +0.000, E1   -36.098, E3 +388884.214}
ENDSPLINE

SPLINE
SPL {X  -162.820, Y  +467.031, Z    +0.000, E1   -36.178, E3 +388903.304}
SPL {X  -162.820, Y  +471.524, Z    +0.000, E1   -36.022, E3 +388916.857}
SPL {X  -162.820, Y  +475.701, Z    +0.000, E1   -36.157, E3 +388928.038}
SPL {X  -162.820, Y  +479.954, Z    +0.000, E1   -36.086, E3 +388940.579}
SPL {X  -162.820, Y  +485.438, Z    +0.000, E1   -36.112, E3 +388956.297}
SPL {X  -162.820, Y  +490.843, Z    +0.000, E1   -36.087, E3 +388971.710}
SPL {X  -162.820, Y  +494.712, Z    +0.000, E1   -36.164, E3 +388982.222}
SPL {X  -162.820, Y  +498.932, Z    +0.000, E1   -36.079, E3 +388994.949}
SPL {X  -162.820, Y  +504.528, Z    +0.000, E1   -36.109, E3 +389010.745}
SPL {X  -162.820, Y  +509.364, Z    +0.000, E1   -36.084, E3 +389024.650}
SPL {X  -162.820, Y  +515.001, Z    +0.000, E1   -36.183, E3 +389040.288}
SPL {X  -162.820, Y  +520.482, Z    +0.000, E1   -36.096, E3 +389056.333}
SPL {X  -162.820, Y  +524.107, Z    +0.000, E1   -36.045, E3 +389066.917}
SPL {X  -162.820, Y  +527.962, Z    +0.000, E1   -36.074, E3 +389077.850}
SPL {X  -162.820, Y  +532.253, Z    +0.000, E1   -36.170, E3 +389089.439}
SPL {X  -162.820, Y  +536.031, Z    +0.000, E1   -36.058, E3 +389100.977}
SPL {X  -162.820, Y  +541.179, Z    +0.000, E1   -36.085, E3 +389115.618}
SPL {X  -162.820, Y  +546.355, Z    +0.000, E1   -36.114, E3 +389130.162}
SPL {X  -162.820, Y  +550.585, Z    +0.000, E1   -36.077, E3 +389142.432}
SPL {X  -162.820, Y  +555.903, Z    +0.000, E1   -36.136, E3 +389157.430}
SPL {X  -162.820, Y  +560.354, Z    +0.000, E1   -36.138, E3 +389169.884}
SPL {X  -162.820, Y  +562.721, Z    +0.000, E1   -36.046, E3 +389177.229}
SPL {X  -162.820, Y  +566.500, Z    +0.000, E1   -36.073, E3 +389187.961}
SPL {X  -162.820, Y  +571.734, Z    +0.000, E1   -36.094, E3 +389202.891}
SPL {X  -162.820, Y  +576.887, Z    +0.000, E1   -36.084, E3 +389217.585}
SPL {X  -162.820, Y  +581.763, Z    +0.000, E1   -36.093, E3 +389231.521}
SPL {X  -162.820, Y  +586.693, Z    +0.000, E1   -36.086, E3 +389245.626}
SPL {X  -162.820, Y  +590.250, Z    +0.000, E1   -36.075, E3 +389255.745}
SPL {X  -162.820, Y  +592.727, Z    +0.000, E1   -35.960, E3 +389263.569}
SPL {X  -162.820, Y  +597.399, Z    +0.000, E1   -36.147, E3 +389275.917}
SPL {X  -162.820, Y  +602.243, Z    +0.000, E1   -36.085, E3 +389290.063}
SPL {X  -162.820, Y  +605.848, Z    +0.000, E1   -36.070, E3 +389300.385}
SPL {X  -162.820, Y  +609.375, Z    +0.000, E1   -36.084, E3 +389310.435}
SPL {X  -162.820, Y  +612.959, Z    +0.000, E1   -36.034, E3 +389320.955}
SPL {X  -162.820, Y  +616.897, Z    +0.000, E1   -36.061, E3 +389332.103}
SPL {X  -162.820, Y  +621.516, Z    +0.000, E1   -36.072, E3 +389345.302}
SPL {X  -162.820, Y  +626.243, Z    +0.000, E1   -36.105, E3 +389358.545}
SPL {X  -162.820, Y  +630.571, Z    +0.000, E1   -36.057, E3 +389371.247}
SPL {X  -162.820, Y  +635.505, Z    +0.000, E1   -36.079, E3 +389385.253}
SPL {X  -162.820, Y  +639.747, Z    +0.000, E1   -36.079, E3 +389397.279}
SPL {X  -162.820, Y  +642.832, Z    +0.000, E1   -36.091, E3 +389406.003}
SPL {X  -162.820, Y  +646.320, Z    +0.000, E1   -36.078, E3 +389416.110}
SPL {X  -162.820, Y  +649.997, Z    +0.000, E1   -36.000, E3 +389427.081}
SPL {X  -162.820, Y  +655.571, Z    +0.000, E1   -36.141, E3 +389442.415}
SPL {X  -162.820, Y  +661.560, Z    +0.000, E1   -36.068, E3 +389459.843}
SPL {X  -162.820, Y  +666.386, Z    +0.000, E1   -36.048, E3 +389473.727}
SPL {X  -162.820, Y  +672.345, Z    +0.000, E1   -36.097, E3 +389490.668}
SPL {X  -162.761, Y  +677.889, Z    +0.000, E1   -36.122, E3 +389506.132}
SPL {X  -162.577, Y  +682.401, Z    +0.000, E1   -36.021, E3 +389519.749}
SPL {X  -162.296, Y  +686.558, Z    +0.000, E1   -35.952, E3 +389531.940}
SPL {X  -161.948, Y  +690.331, Z    +0.000, E1   -35.960, E3 +389542.738}
SPL {X  -161.544, Y  +693.846, Z    +0.000, E1   -35.908, E3 +389553.013}
SPL {X  -161.078, Y  +697.256, Z    +0.000, E1   -35.797, E3 +389563.519}
SPL {X  -160.313, Y  +701.964, Z    +0.000, E1   -35.709, E3 +389577.595}
SPL {X  -159.622, Y  +705.613, Z    +0.000, E1   -35.430, E3 +389589.534}
SPL {X  -158.758, Y  +709.640, Z    +0.000, E1   -35.380, E3 +389601.541}
SPL {X  -155.037, Y  +723.239, Z    +0.000, E1   -39.382, E3 +389614.426}
SPL {X  -152.141, Y  +731.494, Z    +0.000, E1   -35.181, E3 +389673.232}
ENDSPLINE

SPLINE
SPL {X  -160.133, Y  +702.956, Z    +0.000, E1   -19.806, E3 +389716.770}
SPL {X  -161.979, Y  +690.023, Z    +0.000, E1   -12.991, E3 +389719.686}
SPL {X  -162.783, Y  +676.950, Z    +0.000, E1    -5.489, E3 +389720.216}
SPL {X  -162.820, Y  +669.862, Z    +0.000, E1    -0.751, E3 +389722.612}
SPL {X  -162.820, Y  +665.790, Z    +0.000, E1    +2.338, E3 +389721.985}
SPL {X  -162.820, Y  +662.868, Z    +0.000, E1    +4.743, E3 +389723.042}
SPL {X  -162.820, Y  +657.781, Z    +0.000, E1    +9.391, E3 +389720.249}
SPL {X  -162.820, Y  +648.706, Z    +0.000, E1   +17.761, E3 +389722.001}
SPL {X  -162.820, Y  +635.926, Z    +0.000, E1   +28.192, E3 +389726.828}
SPL {X  -162.820, Y  +621.673, Z    +0.000, E1   +34.265, E3 +389743.186}
SPL {X  -162.820, Y  +601.185, Z    +0.000, E1   +39.430, E3 +389769.764}
SPL {X  -162.820, Y  +599.927, Z    +0.000, E1   +35.241, E3 +389796.342}
SPL {X  -162.820, Y  +597.570, Z    +0.000, E1   +33.919, E3 +389812.071}
SPL {X  -162.820, Y  +592.692, Z    +0.000, E1   +33.779, E3 +389827.963}
SPL {X  -162.820, Y  +588.795, Z    +0.000, E1   +33.876, E3 +389839.400}
SPL {X  -162.820, Y  +585.519, Z    +0.000, E1   +33.888, E3 +389849.485}
SPL {X  -162.820, Y  +582.066, Z    +0.000, E1   +33.857, E3 +389860.419}
SPL {X  -162.820, Y  +577.919, Z    +0.000, E1   +33.841, E3 +389873.472}
SPL {X  -162.820, Y  +573.566, Z    +0.000, E1   +33.899, E3 +389886.547}
SPL {X  -162.820, Y  +569.298, Z    +0.000, E1   +33.851, E3 +389900.188}
SPL {X  -162.820, Y  +563.983, Z    +0.000, E1   +33.916, E3 +389916.329}
SPL {X  -162.820, Y  +559.395, Z    +0.000, E1   +33.796, E3 +389931.211}
SPL {X  -162.820, Y  +554.453, Z    +0.000, E1   +33.841, E3 +389946.435}
SPL {X  -162.820, Y  +549.726, Z    +0.000, E1   +33.905, E3 +389960.539}
SPL {X  -162.820, Y  +545.760, Z    +0.000, E1   +33.901, E3 +389972.935}
SPL {X  -162.820, Y  +541.668, Z    +0.000, E1   +33.787, E3 +389986.334}
SPL {X  -162.820, Y  +538.174, Z    +0.000, E1   +33.865, E3 +389996.624}
SPL {X  -162.820, Y  +534.943, Z    +0.000, E1   +33.919, E3 +390006.364}
SPL {X  -162.820, Y  +531.459, Z    +0.000, E1   +33.783, E3 +390018.021}
SPL {X  -162.820, Y  +526.783, Z    +0.000, E1   +33.870, E3 +390032.149}
SPL {X  -162.820, Y  +521.520, Z    +0.000, E1   +33.826, E3 +390048.796}
SPL {X  -162.820, Y  +516.814, Z    +0.000, E1   +33.917, E3 +390062.698}
SPL {X  -162.820, Y  +512.685, Z    +0.000, E1   +33.830, E3 +390076.141}
SPL {X  -162.820, Y  +508.888, Z    +0.000, E1   +33.871, E3 +390087.555}
SPL {X  -162.820, Y  +505.651, Z    +0.000, E1   +33.839, E3 +390097.872}
SPL {X  -162.820, Y  +500.931, Z    +0.000, E1   +34.256, E3 +390109.746}
SPL {X  -162.820, Y  +481.122, Z    +0.000, E1   +41.279, E3 +390120.010}
SPL {X  -162.820, Y  +477.698, Z    +0.000, E1   +40.353, E3 +390134.066}
SPL {X  -162.820, Y  +474.538, Z    +0.000, E1   +39.267, E3 +390148.242}
SPL {X  -162.820, Y  +472.097, Z    +0.000, E1   +38.411, E3 +390159.785}
SPL {X  -162.820, Y  +469.308, Z    +0.000, E1   +37.839, E3 +390170.590}
SPL {X  -162.820, Y  +467.216, Z    +0.000, E1   +37.215, E3 +390180.156}
SPL {X  -162.820, Y  +462.598, Z    +0.000, E1   +37.325, E3 +390192.110}
SPL {X  -162.820, Y  +457.832, Z    +0.000, E1   +37.294, E3 +390205.397}
SPL {X  -162.820, Y  +452.986, Z    +0.000, E1   +37.368, E3 +390218.131}
SPL {X  -162.820, Y  +448.311, Z    +0.000, E1   +37.333, E3 +390231.151}
SPL {X  -162.820, Y  +443.351, Z    +0.000, E1   +37.335, E3 +390244.680}
SPL {X  -162.820, Y  +438.727, Z    +0.000, E1   +37.289, E3 +390257.553}
SPL {X  -162.820, Y  +434.320, Z    +0.000, E1   +37.343, E3 +390269.263}
SPL {X  -162.820, Y  +430.091, Z    +0.000, E1   +37.424, E3 +390280.263}
SPL {X  -162.820, Y  +426.177, Z    +0.000, E1   +37.250, E3 +390292.086}
SPL {X  -162.820, Y  +421.391, Z    +0.000, E1   +37.346, E3 +390304.549}
SPL {X  -162.820, Y  +416.811, Z    +0.000, E1   +37.348, E3 +390317.083}
SPL {X  -162.820, Y  +411.860, Z    +0.000, E1   +37.402, E3 +390330.235}
SPL {X  -162.820, Y  +407.726, Z    +0.000, E1   +37.291, E3 +390342.183}
SPL {X  -162.820, Y  +403.543, Z    +0.000, E1   +37.305, E3 +390353.528}
SPL {X  -162.820, Y  +399.300, Z    +0.000, E1   +37.355, E3 +390364.813}
SPL {X  -162.820, Y  +395.182, Z    +0.000, E1   +37.347, E3 +390376.102}
SPL {X  -162.820, Y  +390.797, Z    +0.000, E1   +37.358, E3 +390388.014}
SPL {X  -162.820, Y  +385.307, Z    +0.000, E1   +37.364, E3 +390403.094}
SPL {X  -162.820, Y  +380.796, Z    +0.000, E1   +37.334, E3 +390415.380}
SPL {X  -162.785, Y  +377.133, Z    +0.000, E1   +37.299, E3 +390425.701}
SPL {X  -162.623, Y  +372.484, Z    +0.000, E1   +37.337, E3 +390438.141}
SPL {X  -162.331, Y  +367.894, Z    +0.000, E1   +37.251, E3 +390451.254}
SPL {X  -161.920, Y  +363.407, Z    +0.000, E1   +37.164, E3 +390463.988}
SPL {X  -161.341, Y  +358.603, Z    +0.000, E1   +37.117, E3 +390477.468}
SPL {X  -160.616, Y  +353.801, Z    +0.000, E1   +36.942, E3 +390491.632}
SPL {X  -159.837, Y  +349.474, Z    +0.000, E1   +36.824, E3 +390504.077}
SPL {X  -158.862, Y  +344.820, Z    +0.000, E1   +36.732, E3 +390517.439}
SPL {X  -157.959, Y  +341.011, Z    +0.000, E1   +36.448, E3 +390529.336}
SPL {X  -154.495, Y  +329.104, Z    +0.000, E1   +40.891, E3 +390534.219}
SPL {X  -152.543, Y  +323.569, Z    +0.000, E1   +41.772, E3 +390541.975}
SPL {X  -150.942, Y  +319.452, Z    +0.000, E1   +36.529, E3 +390594.525}
ENDSPLINE

SPLINE
SPL {X  -159.264, Y  +346.659, Z    +0.000, E1   +22.083, E3 +390635.099}
SPL {X  -161.245, Y  +357.907, Z    +0.000, E1   +16.095, E3 +390648.532}
SPL {X  -162.697, Y  +374.161, Z    +0.000, E1    +7.119, E3 +390646.522}
SPL {X  -162.820, Y  +380.878, Z    +0.000, E1    +2.854, E3 +390649.353}
SPL {X  -162.820, Y  +385.313, Z    +0.000, E1    -0.228, E3 +390649.133}
SPL {X  -162.820, Y  +389.965, Z    +0.000, E1    -3.918, E3 +390648.502}
SPL {X  -162.820, Y  +394.532, Z    +0.000, E1    -7.849, E3 +390650.050}
SPL {X  -162.820, Y  +400.765, Z    +0.000, E1   -14.108, E3 +390647.517}
SPL {X  -162.820, Y  +411.829, Z    +0.000, E1   -24.195, E3 +390649.594}
SPL {X  -162.820, Y  +434.900, Z    +0.000, E1   -34.666, E3 +390676.959}
SPL {X  -162.820, Y  +465.440, Z    +0.000, E1   -41.264, E3 +390718.266}
ENDSPLINE

SPLINE
SPL {X  -162.820, Y  +460.175, Z    +0.000, E1   -36.098, E3 +390736.066}
ENDSPLINE

SPLINE
SPL {X  -162.820, Y  +467.031, Z    +0.000, E1   -36.178, E3 +390755.156}
SPL {X  -162.820, Y  +471.524, Z    +0.000, E1   -36.022, E3 +390768.709}
SPL {X  -162.820, Y  +475.701, Z    +0.000, E1   -36.157, E3 +390779.890}
SPL {X  -162.820, Y  +479.954, Z    +0.000, E1   -36.086, E3 +390792.430}
SPL {X  -162.820, Y  +485.438, Z    +0.000, E1   -36.112, E3 +390808.149}
SPL {X  -162.820, Y  +490.843, Z    +0.000, E1   -36.087, E3 +390823.562}
SPL {X  -162.820, Y  +494.712, Z    +0.000, E1   -36.164, E3 +390834.074}
SPL {X  -162.820, Y  +497.796, Z    +0.000, E1   -36.022, E3 +390843.780}
SPL {X  -162.820, Y  +502.146, Z    +0.000, E1   -36.123, E3 +390855.649}
SPL {X  -162.820, Y  +505.688, Z    +0.000, E1   -36.050, E3 +390866.131}
SPL {X  -162.820, Y  +509.364, Z    +0.000, E1   -36.084, E3 +390876.502}
SPL {X  -162.820, Y  +515.001, Z    +0.000, E1   -36.183, E3 +390892.140}
SPL {X  -162.820, Y  +520.482, Z    +0.000, E1   -36.096, E3 +390908.185}
SPL {X  -162.820, Y  +524.107, Z    +0.000, E1   -36.045, E3 +390918.769}
SPL {X  -162.820, Y  +527.962, Z    +0.000, E1   -36.074, E3 +390929.702}
SPL {X  -162.820, Y  +532.253, Z    +0.000, E1   -36.170, E3 +390941.291}
SPL {X  -162.820, Y  +536.031, Z    +0.000, E1   -36.058, E3 +390952.829}
SPL {X  -162.820, Y  +540.096, Z    +0.000, E1   -36.040, E3 +390964.527}
SPL {X  -162.820, Y  +545.472, Z    +0.000, E1   -36.142, E3 +390979.465}
SPL {X  -162.820, Y  +550.585, Z    +0.000, E1   -36.077, E3 +390994.283}
SPL {X  -162.820, Y  +555.903, Z    +0.000, E1   -36.136, E3 +391009.282}
SPL {X  -162.820, Y  +561.684, Z    +0.000, E1   -36.118, E3 +391025.811}
SPL {X  -162.820, Y  +566.500, Z    +0.000, E1   -36.073, E3 +391039.813}
SPL {X  -162.820, Y  +571.734, Z    +0.000, E1   -36.094, E3 +391054.743}
SPL {X  -162.820, Y  +578.070, Z    +0.000, E1   -36.120, E3 +391072.759}
SPL {X  -162.820, Y  +582.838, Z    +0.000, E1   -36.064, E3 +391086.503}
SPL {X  -162.820, Y  +586.693, Z    +0.000, E1   -36.086, E3 +391097.478}
SPL {X  -162.820, Y  +591.665, Z    +0.000, E1   -36.045, E3 +391112.006}
SPL {X  -162.820, Y  +597.399, Z    +0.000, E1   -36.147, E3 +391127.769}
SPL {X  -162.820, Y  +602.243, Z    +0.000, E1   -36.085, E3 +391141.915}
SPL {X  -162.820, Y  +605.848, Z    +0.000, E1   -36.070, E3 +391152.237}
SPL {X  -162.820, Y  +609.375, Z    +0.000, E1   -36.084, E3 +391162.287}
SPL {X  -162.820, Y  +612.959, Z    +0.000, E1   -36.034, E3 +391172.807}
SPL {X  -162.820, Y  +616.897, Z    +0.000, E1   -36.061, E3 +391183.955}
SPL {X  -162.820, Y  +620.590, Z    +0.000, E1   -36.079, E3 +391194.350}
SPL {X  -162.820, Y  +625.276, Z    +0.000, E1   -36.104, E3 +391207.766}
SPL {X  -162.820, Y  +630.571, Z    +0.000, E1   -36.057, E3 +391223.099}
SPL {X  -162.820, Y  +635.505, Z    +0.000, E1   -36.079, E3 +391237.104}
SPL {X  -162.820, Y  +641.277, Z    +0.000, E1   -36.126, E3 +391253.397}
SPL {X  -162.820, Y  +646.320, Z    +0.000, E1   -36.078, E3 +391267.962}
SPL {X  -162.820, Y  +651.289, Z    +0.000, E1   -36.059, E3 +391282.419}
SPL {X  -162.820, Y  +656.677, Z    +0.000, E1   -36.110, E3 +391297.432}
SPL {X  -162.820, Y  +660.489, Z    +0.000, E1   -36.068, E3 +391308.498}
SPL {X  -162.820, Y  +665.459, Z    +0.000, E1   -36.068, E3 +391322.944}
SPL {X  -162.820, Y  +671.104, Z    +0.000, E1   -36.061, E3 +391338.998}
SPL {X  -162.787, Y  +676.764, Z    +0.000, E1   -36.126, E3 +391354.898}
SPL {X  -162.577, Y  +682.401, Z    +0.000, E1   -36.021, E3 +391371.601}
SPL {X  -162.187, Y  +687.846, Z    +0.000, E1   -36.007, E3 +391387.270}
SPL {X  -161.667, Y  +692.839, Z    +0.000, E1   -35.918, E3 +391402.035}
SPL {X  -160.925, Y  +698.267, Z    +0.000, E1   -35.816, E3 +391418.297}
SPL {X  -160.151, Y  +702.861, Z    +0.000, E1   -35.643, E3 +391432.267}
SPL {X  -159.622, Y  +705.613, Z    +0.000, E1   -35.430, E3 +391441.386}
SPL {X  -158.758, Y  +709.640, Z    +0.000, E1   -35.380, E3 +391453.393}
SPL {X  -155.037, Y  +723.239, Z    +0.000, E1   -39.382, E3 +391466.278}
SPL {X  -152.141, Y  +731.494, Z    +0.000, E1   -35.181, E3 +391525.084}
ENDSPLINE

SPLINE
SPL {X  -160.133, Y  +702.956, Z    +0.000, E1   -19.806, E3 +391568.622}
SPL {X  -161.979, Y  +690.023, Z    +0.000, E1   -12.991, E3 +391571.538}
SPL {X  -162.641, Y  +681.139, Z    +0.000, E1    -7.893, E3 +391573.630}
SPL {X  -162.820, Y  +673.062, Z    +0.000, E1    -2.992, E3 +391572.597}
SPL {X  -162.820, Y  +666.731, Z    +0.000, E1    +1.545, E3 +391574.227}
SPL {X  -162.820, Y  +660.758, Z    +0.000, E1    +6.523, E3 +391573.938}
SPL {X  -162.820, Y  +650.583, Z    +0.000, E1   +16.035, E3 +391572.910}
SPL {X  -162.820, Y  +629.267, Z    +0.000, E1   +31.872, E3 +391584.059}
SPL {X  -162.820, Y  +620.680, Z    +0.000, E1   +34.107, E3 +391598.108}
SPL {X  -162.820, Y  +609.002, Z    +0.000, E1   +38.458, E3 +391608.259}
SPL {X  -162.820, Y  +596.392, Z    +0.000, E1   +37.895, E3 +391641.728}
ENDSPLINE

SPLINE
SPL {X  -162.820, Y  +599.924, Z    +0.000, E1   +33.992, E3 +391656.102}
ENDSPLINE

SPLINE
SPL {X  -162.820, Y  +595.170, Z    +0.000, E1   +33.784, E3 +391672.150}
SPL {X  -162.820, Y  +589.785, Z    +0.000, E1   +33.904, E3 +391688.147}
SPL {X  -162.820, Y  +584.646, Z    +0.000, E1   +33.882, E3 +391704.216}
SPL {X  -162.820, Y  +579.919, Z    +0.000, E1   +33.857, E3 +391719.004}
SPL {X  -162.820, Y  +574.615, Z    +0.000, E1   +33.920, E3 +391735.178}
SPL {X  -162.820, Y  +570.335, Z    +0.000, E1   +33.821, E3 +391748.884}
SPL {X  -162.820, Y  +565.901, Z    +0.000, E1   +33.889, E3 +391762.404}
SPL {X  -162.820, Y  +560.226, Z    +0.000, E1   +33.868, E3 +391780.190}
SPL {X  -162.820, Y  +554.453, Z    +0.000, E1   +33.841, E3 +391798.287}
SPL {X  -162.820, Y  +549.726, Z    +0.000, E1   +33.905, E3 +391812.390}
SPL {X  -162.820, Y  +545.760, Z    +0.000, E1   +33.901, E3 +391824.786}
SPL {X  -162.820, Y  +541.668, Z    +0.000, E1   +33.787, E3 +391838.186}
SPL {X  -162.820, Y  +538.174, Z    +0.000, E1   +33.865, E3 +391848.476}
SPL {X  -162.820, Y  +534.943, Z    +0.000, E1   +33.919, E3 +391858.216}
SPL {X  -162.820, Y  +530.273, Z    +0.000, E1   +33.855, E3 +391873.245}
SPL {X  -162.820, Y  +524.900, Z    +0.000, E1   +33.820, E3 +391890.146}
SPL {X  -162.820, Y  +520.532, Z    +0.000, E1   +33.805, E3 +391903.714}
SPL {X  -162.820, Y  +516.814, Z    +0.000, E1   +33.917, E3 +391914.550}
SPL {X  -162.820, Y  +512.685, Z    +0.000, E1   +33.830, E3 +391927.992}
SPL {X  -162.820, Y  +508.888, Z    +0.000, E1   +33.871, E3 +391939.407}
SPL {X  -162.820, Y  +505.651, Z    +0.000, E1   +33.839, E3 +391949.724}
SPL {X  -162.820, Y  +500.931, Z    +0.000, E1   +34.256, E3 +391961.598}
SPL {X  -162.820, Y  +481.122, Z    +0.000, E1   +41.279, E3 +391971.862}
SPL {X  -162.820, Y  +478.698, Z    +0.000, E1   +40.526, E3 +391982.211}
SPL {X  -162.820, Y  +475.203, Z    +0.000, E1   +39.596, E3 +391996.671}
SPL {X  -162.820, Y  +472.097, Z    +0.000, E1   +38.411, E3 +392011.637}
SPL {X  -162.820, Y  +469.308, Z    +0.000, E1   +37.839, E3 +392022.441}
SPL {X  -162.820, Y  +467.216, Z    +0.000, E1   +37.215, E3 +392032.008}
SPL {X  -162.820, Y  +462.598, Z    +0.000, E1   +37.325, E3 +392043.962}
SPL {X  -162.820, Y  +457.832, Z    +0.000, E1   +37.294, E3 +392057.249}
SPL {X  -162.820, Y  +452.986, Z    +0.000, E1   +37.368, E3 +392069.983}
SPL {X  -162.820, Y  +448.311, Z    +0.000, E1   +37.333, E3 +392083.003}
SPL {X  -162.820, Y  +443.351, Z    +0.000, E1   +37.335, E3 +392096.532}
SPL {X  -162.820, Y  +438.727, Z    +0.000, E1   +37.289, E3 +392109.405}
SPL {X  -162.820, Y  +434.320, Z    +0.000, E1   +37.343, E3 +392121.115}
SPL {X  -162.820, Y  +430.091, Z    +0.000, E1   +37.424, E3 +392132.115}
SPL {X  -162.820, Y  +426.177, Z    +0.000, E1   +37.250, E3 +392143.937}
SPL {X  -162.820, Y  +420.241, Z    +0.000, E1   +37.355, E3 +392159.644}
SPL {X  -162.820, Y  +415.595, Z    +0.000, E1   +37.375, E3 +392171.984}
SPL {X  -162.820, Y  +411.860, Z    +0.000, E1   +37.402, E3 +392182.087}
SPL {X  -162.820, Y  +407.726, Z    +0.000, E1   +37.291, E3 +392194.035}
SPL {X  -162.820, Y  +403.543, Z    +0.000, E1   +37.305, E3 +392205.380}
SPL {X  -162.820, Y  +399.300, Z    +0.000, E1   +37.355, E3 +392216.664}
SPL {X  -162.820, Y  +395.182, Z    +0.000, E1   +37.347, E3 +392227.954}
SPL {X  -162.820, Y  +390.797, Z    +0.000, E1   +37.358, E3 +392239.866}
SPL {X  -162.820, Y  +386.671, Z    +0.000, E1   +37.363, E3 +392251.047}
SPL {X  -162.820, Y  +382.174, Z    +0.000, E1   +37.329, E3 +392263.624}
SPL {X  -162.785, Y  +377.133, Z    +0.000, E1   +37.299, E3 +392277.553}
SPL {X  -162.623, Y  +372.484, Z    +0.000, E1   +37.337, E3 +392289.993}
SPL {X  -162.331, Y  +367.894, Z    +0.000, E1   +37.251, E3 +392303.106}
SPL {X  -161.920, Y  +363.407, Z    +0.000, E1   +37.164, E3 +392315.840}
SPL {X  -161.482, Y  +359.669, Z    +0.000, E1   +37.064, E3 +392326.624}
SPL {X  -160.943, Y  +355.851, Z    +0.000, E1   +37.136, E3 +392336.611}
SPL {X  -160.493, Y  +353.069, Z    +0.000, E1   +36.789, E3 +392346.263}
SPL {X  -159.837, Y  +349.474, Z    +0.000, E1   +36.824, E3 +392355.929}
SPL {X  -159.171, Y  +346.224, Z    +0.000, E1   +36.747, E3 +392365.205}
SPL {X  -158.248, Y  +342.188, Z    +0.000, E1   +36.583, E3 +392377.368}
SPL {X  -153.520, Y  +326.260, Z    +0.000, E1   +41.363, E3 +392390.020}
SPL {X  -150.942, Y  +319.452, Z    +0.000, E1   +36.529, E3 +392446.377}
ENDSPLINE

SPLINE
SPL {X  -159.264, Y  +346.659, Z    +0.000, E1   +22.083, E3 +392486.951}
SPL {X  -161.245, Y  +357.907, Z    +0.000, E1   +16.095, E3 +392500.384}
SPL {X  -162.746, Y  +375.590, Z    +0.000, E1    +6.280, E3 +392499.972}
SPL {X  -162.820, Y  +384.478, Z    +0.000, E1    +0.434, E3 +392500.642}
SPL {X  -162.820, Y  +389.965, Z    +0.000, E1    -3.918, E3 +392500.353}
SPL {X  -162.820, Y  +394.532, Z    +0.000, E1    -7.849, E3 +392501.902}
SPL {X  -162.820, Y  +400.765, Z    +0.000, E1   -14.108, E3 +392499.368}
SPL {X  -162.820, Y  +411.829, Z    +0.000, E1   -24.195, E3 +392501.446}
SPL {X  -162.820, Y  +434.900, Z    +0.000, E1   -34.666, E3 +392528.811}
SPL {X  -162.820, Y  +465.440, Z    +0.000, E1   -41.264, E3 +392570.118}
ENDSPLINE

SPLINE
SPL {X  -162.820, Y  +460.175, Z    +0.000, E1   -36.098, E3 +392587.918}
ENDSPLINE

SPLINE
SPL {X  -162.820, Y  +465.690, Z    +0.000, E1   -36.140, E3 +392603.232}
SPL {X  -162.820, Y  +470.432, Z    +0.000, E1   -36.100, E3 +392617.114}
SPL {X  -162.820, Y  +475.701, Z    +0.000, E1   -36.157, E3 +392631.742}
SPL {X  -162.820, Y  +479.954, Z    +0.000, E1   -36.086, E3 +392644.282}
SPL {X  -162.820, Y  +483.976, Z    +0.000, E1   -36.049, E3 +392656.014}
SPL {X  -162.820, Y  +488.601, Z    +0.000, E1   -36.081, E3 +392669.104}
SPL {X  -162.820, Y  +493.837, Z    +0.000, E1   -36.178, E3 +392683.448}
SPL {X  -162.820, Y  +497.796, Z    +0.000, E1   -36.022, E3 +392695.632}
SPL {X  -162.820, Y  +502.146, Z    +0.000, E1   -36.123, E3 +392707.501}
SPL {X  -162.820, Y  +505.688, Z    +0.000, E1   -36.050, E3 +392717.983}
SPL {X  -162.820, Y  +509.364, Z    +0.000, E1   -36.084, E3 +392728.354}
SPL {X  -162.820, Y  +515.001, Z    +0.000, E1   -36.183, E3 +392743.991}
SPL {X  -162.820, Y  +520.482, Z    +0.000, E1   -36.096, E3 +392760.037}
SPL {X  -162.820, Y  +524.107, Z    +0.000, E1   -36.045, E3 +392770.621}
SPL {X  -162.820, Y  +527.962, Z    +0.000, E1   -36.074, E3 +392781.554}
SPL {X  -162.820, Y  +532.253, Z    +0.000, E1   -36.170, E3 +392793.143}
SPL {X  -162.820, Y  +536.031, Z    +0.000, E1   -36.058, E3 +392804.681}
SPL {X  -162.820, Y  +541.179, Z    +0.000, E1   -36.085, E3 +392819.322}
SPL {X  -162.820, Y  +546.355, Z    +0.000, E1   -36.114, E3 +392833.866}
SPL {X  -162.820, Y  +550.585, Z    +0.000, E1   -36.077, E3 +392846.135}
SPL {X  -162.820, Y  +555.903, Z    +0.000, E1   -36.136, E3 +392861.134}
SPL {X  -162.820, Y  +560.354, Z    +0.000, E1   -36.138, E3 +392873.587}
SPL {X  -162.820, Y  +562.721, Z    +0.000, E1   -36.046, E3 +392880.933}
SPL {X  -162.820, Y  +566.500, Z    +0.000, E1   -36.073, E3 +392891.665}
SPL {X  -162.820, Y  +570.319, Z    +0.000, E1   -36.045, E3 +392902.693}
SPL {X  -162.820, Y  +573.265, Z    +0.000, E1   -36.071, E3 +392910.930}
SPL {X  -162.820, Y  +578.070, Z    +0.000, E1   -36.120, E3 +392924.611}
SPL {X  -162.820, Y  +582.838, Z    +0.000, E1   -36.064, E3 +392938.354}
SPL {X  -162.820, Y  +586.693, Z    +0.000, E1   -36.086, E3 +392949.330}
SPL {X  -162.820, Y  +591.665, Z    +0.000, E1   -36.045, E3 +392963.858}
SPL {X  -162.820, Y  +596.059, Z    +0.000, E1   -36.124, E3 +392975.790}
SPL {X  -162.820, Y  +598.788, Z    +0.000, E1   -36.102, E3 +392983.701}
SPL {X  -162.820, Y  +602.243, Z    +0.000, E1   -36.085, E3 +392993.767}
SPL {X  -162.820, Y  +605.848, Z    +0.000, E1   -36.070, E3 +393004.088}
SPL {X  -162.820, Y  +609.375, Z    +0.000, E1   -36.084, E3 +393014.139}
SPL {X  -162.820, Y  +612.959, Z    +0.000, E1   -36.034, E3 +393024.659}
SPL {X  -162.820, Y  +616.897, Z    +0.000, E1   -36.061, E3 +393035.807}
SPL {X  -162.820, Y  +621.516, Z    +0.000, E1   -36.072, E3 +393049.006}
SPL {X  -162.820, Y  +626.243, Z    +0.000, E1   -36.105, E3 +393062.248}
SPL {X  -162.820, Y  +630.571, Z    +0.000, E1   -36.057, E3 +393074.950}
SPL {X  -162.820, Y  +635.505, Z    +0.000, E1   -36.079, E3 +393088.956}
SPL {X  -162.820, Y  +639.747, Z    +0.000, E1   -36.079, E3 +393100.983}
SPL {X  -162.820, Y  +642.832, Z    +0.000, E1   -36.091, E3 +393109.707}
SPL {X  -162.820, Y  +646.320, Z    +0.000, E1   -36.078, E3 +393119.814}
SPL {X  -162.820, Y  +651.289, Z    +0.000, E1   -36.059, E3 +393134.270}
SPL {X  -162.820, Y  +656.677, Z    +0.000, E1   -36.110, E3 +393149.284}
SPL {X  -162.820, Y  +661.560, Z    +0.000, E1   -36.068, E3 +393163.547}
SPL {X  -162.820, Y  +666.386, Z    +0.000, E1   -36.048, E3 +393177.431}
SPL {X  -162.820, Y  +672.345, Z    +0.000, E1   -36.097, E3 +393194.372}
SPL {X  -162.761, Y  +677.889, Z    +0.000, E1   -36.122, E3 +393209.836}
SPL {X  -162.577, Y  +682.401, Z    +0.000, E1   -36.021, E3 +393223.453}
SPL {X  -162.187, Y  +687.846, Z    +0.000, E1   -36.007, E3 +393239.122}
SPL {X  -161.667, Y  +692.839, Z    +0.000, E1   -35.918, E3 +393253.887}
SPL {X  -161.078, Y  +697.256, Z    +0.000, E1   -35.797, E3 +393267.223}
SPL {X  -160.313, Y  +701.964, Z    +0.000, E1   -35.709, E3 +393281.298}
SPL {X  -159.317, Y  +707.091, Z    +0.000, E1   -35.482, E3 +393297.322}
SPL {X  -158.510, Y  +710.714, Z    +0.000, E1   -35.230, E3 +393309.033}
SPL {X  -155.037, Y  +723.239, Z    +0.000, E1   -39.382, E3 +393318.130}
SPL {X  -152.141, Y  +731.494, Z    +0.000, E1   -35.181, E3 +393376.935}
ENDSPLINE

SPLINE
SPL {X  -160.133, Y  +702.956, Z    +0.000, E1   -19.806, E3 +393420.473}
SPL {X  -161.979, Y  +690.023, Z    +0.000, E1   -12.991, E3 +393423.390}
SPL {X  -162.641, Y  +681.139, Z    +0.000, E1    -7.893, E3 +393425.482}
SPL {X  -162.815, Y  +674.833, Z    +0.000, E1    -4.093, E3 +393423.098}
SPL {X  -162.820, Y  +669.862, Z    +0.000, E1    -0.751, E3 +393426.316}
SPL {X  -162.820, Y  +665.790, Z    +0.000, E1    +2.338, E3 +393425.688}
SPL {X  -162.820, Y  +660.758, Z    +0.000, E1    +6.523, E3 +393425.789}
SPL {X  -162.820, Y  +655.722, Z    +0.000, E1   +11.608, E3 +393422.162}
SPL {X  -162.820, Y  +648.706, Z    +0.000, E1   +17.761, E3 +393425.704}
SPL {X  -162.820, Y  +635.926, Z    +0.000, E1   +28.192, E3 +393430.532}
SPL {X  -162.820, Y  +621.673, Z    +0.000, E1   +34.265, E3 +393446.889}
SPL {X  -162.820, Y  +609.002, Z    +0.000, E1   +38.458, E3 +393460.111}
SPL {X  -162.820, Y  +596.392, Z    +0.000, E1   +37.895, E3 +393493.580}
ENDSPLINE

SPLINE
SPL {X  -162.820, Y  +599.924, Z    +0.000, E1   +33.992, E3 +393507.954}
ENDSPLINE

SPLINE
SPL {X  -162.820, Y  +596.128, Z    +0.000, E1   +33.827, E3 +393520.591}
SPL {X  -162.820, Y  +592.692, Z    +0.000, E1   +33.779, E3 +393531.667}
SPL {X  -162.820, Y  +588.795, Z    +0.000, E1   +33.876, E3 +393543.104}
SPL {X  -162.820, Y  +584.646, Z    +0.000, E1   +33.882, E3 +393556.068}
SPL {X  -162.820, Y  +579.919, Z    +0.000, E1   +33.857, E3 +393570.856}
SPL {X  -162.820, Y  +576.636, Z    +0.000, E1   +33.845, E3 +393581.002}
SPL {X  -162.820, Y  +573.566, Z    +0.000, E1   +33.899, E3 +393590.251}
SPL {X  -162.820, Y  +570.335, Z    +0.000, E1   +33.821, E3 +393600.736}
SPL {X  -162.820, Y  +565.901, Z    +0.000, E1   +33.889, E3 +393614.256}
SPL {X  -162.820, Y  +562.173, Z    +0.000, E1   +33.897, E3 +393625.547}
SPL {X  -162.820, Y  +558.179, Z    +0.000, E1   +33.857, E3 +393638.482}
SPL {X  -162.820, Y  +553.486, Z    +0.000, E1   +33.777, E3 +393653.388}
SPL {X  -162.820, Y  +548.576, Z    +0.000, E1   +33.950, E3 +393667.669}
SPL {X  -162.820, Y  +544.808, Z    +0.000, E1   +33.827, E3 +393679.932}
SPL {X  -162.820, Y  +541.668, Z    +0.000, E1   +33.787, E3 +393690.038}
SPL {X  -162.820, Y  +538.174, Z    +0.000, E1   +33.865, E3 +393700.328}
SPL {X  -162.820, Y  +534.943, Z    +0.000, E1   +33.919, E3 +393710.068}
SPL {X  -162.820, Y  +531.459, Z    +0.000, E1   +33.783, E3 +393721.725}
SPL {X  -162.820, Y  +528.475, Z    +0.000, E1   +33.876, E3 +393730.339}
SPL {X  -162.820, Y  +524.900, Z    +0.000, E1   +33.820, E3 +393741.998}
SPL {X  -162.820, Y  +520.532, Z    +0.000, E1   +33.805, E3 +393755.565}
SPL {X  -162.820, Y  +516.814, Z    +0.000, E1   +33.917, E3 +393766.401}
SPL {X  -162.820, Y  +512.685, Z    +0.000, E1   +33.830, E3 +393779.844}
SPL {X  -162.820, Y  +508.888, Z    +0.000, E1   +33.871, E3 +393791.259}
SPL {X  -162.820, Y  +505.651, Z    +0.000, E1   +33.839, E3 +393801.576}
SPL {X  -162.820, Y  +500.931, Z    +0.000, E1   +34.256, E3 +393813.450}
SPL {X  -162.820, Y  +481.122, Z    +0.000, E1   +41.279, E3 +393823.714}
SPL {X  -162.820, Y  +478.698, Z    +0.000, E1   +40.526, E3 +393834.063}
SPL {X  -162.820, Y  +476.364, Z    +0.000, E1   +39.976, E3 +393843.024}
SPL {X  -162.820, Y  +473.851, Z    +0.000, E1   +39.059, E3 +393855.161}
SPL {X  -162.820, Y  +470.157, Z    +0.000, E1   +38.016, E3 +393871.098}
SPL {X  -162.820, Y  +467.216, Z    +0.000, E1   +37.215, E3 +393883.860}
SPL {X  -162.820, Y  +462.598, Z    +0.000, E1   +37.325, E3 +393895.814}
SPL {X  -162.820, Y  +459.177, Z    +0.000, E1   +37.207, E3 +393905.841}
SPL {X  -162.820, Y  +453.939, Z    +0.000, E1   +37.397, E3 +393919.194}
SPL {X  -162.820, Y  +448.311, Z    +0.000, E1   +37.333, E3 +393934.854}
SPL {X  -162.820, Y  +443.351, Z    +0.000, E1   +37.335, E3 +393948.384}
SPL {X  -162.820, Y  +438.727, Z    +0.000, E1   +37.289, E3 +393961.256}
SPL {X  -162.820, Y  +434.320, Z    +0.000, E1   +37.343, E3 +393972.966}
SPL {X  -162.820, Y  +430.091, Z    +0.000, E1   +37.424, E3 +393983.966}
SPL {X  -162.820, Y  +426.177, Z    +0.000, E1   +37.250, E3 +393995.789}
SPL {X  -162.820, Y  +420.241, Z    +0.000, E1   +37.355, E3 +394011.496}
SPL {X  -162.820, Y  +415.595, Z    +0.000, E1   +37.375, E3 +394023.836}
SPL {X  -162.820, Y  +411.860, Z    +0.000, E1   +37.402, E3 +394033.939}
SPL {X  -162.820, Y  +407.726, Z    +0.000, E1   +37.291, E3 +394045.887}
SPL {X  -162.820, Y  +403.543, Z    +0.000, E1   +37.305, E3 +394057.232}
SPL {X  -162.820, Y  +399.300, Z    +0.000, E1   +37.355, E3 +394068.516}
SPL {X  -162.820, Y  +395.182, Z    +0.000, E1   +37.347, E3 +394079.805}
SPL {X  -162.820, Y  +390.797, Z    +0.000, E1   +37.358, E3 +394091.718}
SPL {X  -162.820, Y  +386.671, Z    +0.000, E1   +37.363, E3 +394102.899}
SPL {X  -162.820, Y  +382.174, Z    +0.000, E1   +37.329, E3 +394115.476}
SPL {X  -162.785, Y  +377.133, Z    +0.000, E1   +37.299, E3 +394129.405}
SPL {X  -162.576, Y  +371.586, Z    +0.000, E1   +37.322, E3 +394144.518}
SPL {X  -162.256, Y  +366.963, Z    +0.000, E1   +37.251, E3 +394157.406}
SPL {X  -161.920, Y  +363.407, Z    +0.000, E1   +37.164, E3 +394167.691}
SPL {X  -161.482, Y  +359.669, Z    +0.000, E1   +37.064, E3 +394178.476}
SPL {X  -160.943, Y  +355.851, Z    +0.000, E1   +37.136, E3 +394188.463}
SPL {X  -160.493, Y  +353.069, Z    +0.000, E1   +36.789, E3 +394198.115}
SPL {X  -159.837, Y  +349.474, Z    +0.000, E1   +36.824, E3 +394207.780}
SPL {X  -158.862, Y  +344.820, Z    +0.000, E1   +36.732, E3 +394221.143}
SPL {X  -157.959, Y  +341.011, Z    +0.000, E1   +36.448, E3 +394233.040}
SPL {X  -154.495, Y  +329.104, Z    +0.000, E1   +40.891, E3 +394237.922}
SPL {X  -152.543, Y  +323.569, Z    +0.000, E1   +41.772, E3 +394245.679}
SPL {X  -150.942, Y  +319.452, Z    +0.000, E1   +36.529, E3 +394298.229}
ENDSPLINE

SPLINE
SPL {X  -159.264, Y  +346.659, Z    +0.000, E1   +22.083, E3 +394338.803}
SPL {X  -161.245, Y  +357.907, Z    +0.000, E1   +16.095, E3 +394352.236}
SPL {X  -162.697, Y  +374.161, Z    +0.000, E1    +7.119, E3 +394350.225}
SPL {X  -162.820, Y  +380.878, Z    +0.000, E1    +2.854, E3 +394353.057}
SPL {X  -162.820, Y  +385.313, Z    +0.000, E1    -0.228, E3 +394352.837}
SPL {X  -162.820, Y  +389.965, Z    +0.000, E1    -3.918, E3 +394352.205}
SPL {X  -162.820, Y  +394.532, Z    +0.000, E1    -7.849, E3 +394353.753}
SPL {X  -162.820, Y  +400.765, Z    +0.000, E1   -14.108, E3 +394351.220}
SPL {X  -162.820, Y  +411.829, Z    +0.000, E1   -24.195, E3 +394353.298}
SPL {X  -162.820, Y  +434.900, Z    +0.000, E1   -34.666, E3 +394380.662}
SPL {X  -162.820, Y  +465.440, Z    +0.000, E1   -41.264, E3 +394421.970}
ENDSPLINE

SPLINE
SPL {X  -162.820, Y  +458.794, Z    +0.000, E1   -36.100, E3 +394435.593}
ENDSPLINE

SPLINE
SPL {X  -162.820, Y  +461.779, Z    +0.000, E1   -35.988, E3 +394444.789}
SPL {X  -162.820, Y  +465.690, Z    +0.000, E1   -36.140, E3 +394455.084}
SPL {X  -162.820, Y  +470.432, Z    +0.000, E1   -36.100, E3 +394468.966}
SPL {X  -162.820, Y  +475.701, Z    +0.000, E1   -36.157, E3 +394483.594}
SPL {X  -162.820, Y  +479.954, Z    +0.000, E1   -36.086, E3 +394496.134}
SPL {X  -162.820, Y  +483.976, Z    +0.000, E1   -36.049, E3 +394507.866}
SPL {X  -162.820, Y  +489.628, Z    +0.000, E1   -36.135, E3 +394523.697}
SPL {X  -162.820, Y  +494.712, Z    +0.000, E1   -36.164, E3 +394537.778}
SPL {X  -162.820, Y  +497.796, Z    +0.000, E1   -36.022, E3 +394547.484}
SPL {X  -162.820, Y  +502.146, Z    +0.000, E1   -36.123, E3 +394559.353}
SPL {X  -162.820, Y  +505.688, Z    +0.000, E1   -36.050, E3 +394569.835}
SPL {X  -162.820, Y  +509.364, Z    +0.000, E1   -36.084, E3 +394580.206}
SPL {X  -162.820, Y  +515.001, Z    +0.000, E1   -36.183, E3 +394595.843}
SPL {X  -162.820, Y  +520.482, Z    +0.000, E1   -36.096, E3 +394611.889}
SPL {X  -162.820, Y  +524.107, Z    +0.000, E1   -36.045, E3 +394622.473}
SPL {X  -162.820, Y  +527.962, Z    +0.000, E1   -36.074, E3 +394633.406}
SPL {X  -162.820, Y  +532.253, Z    +0.000, E1   -36.170, E3 +394644.995}
SPL {X  -162.820, Y  +536.031, Z    +0.000, E1   -36.058, E3 +394656.533}
SPL {X  -162.820, Y  +541.179, Z    +0.000, E1   -36.085, E3 +394671.173}
SPL {X  -162.820, Y  +546.355, Z    +0.000, E1   -36.114, E3 +394685.718}
SPL {X  -162.820, Y  +550.585, Z    +0.000, E1   -36.077, E3 +394697.987}
SPL {X  -162.820, Y  +555.903, Z    +0.000, E1   -36.136, E3 +394712.985}
SPL {X  -162.820, Y  +560.354, Z    +0.000, E1   -36.138, E3 +394725.439}
SPL {X  -162.820, Y  +562.721, Z    +0.000, E1   -36.046, E3 +394732.785}
SPL {X  -162.820, Y  +566.500, Z    +0.000, E1   -36.073, E3 +394743.517}
SPL {X  -162.820, Y  +571.734, Z    +0.000, E1   -36.094, E3 +394758.447}
SPL {X  -162.820, Y  +576.887, Z    +0.000, E1   -36.084, E3 +394773.140}
SPL {X  -162.820, Y  +581.763, Z    +0.000, E1   -36.093, E3 +394787.077}
SPL {X  -162.820, Y  +586.693, Z    +0.000, E1   -36.086, E3 +394801.182}
SPL {X  -162.820, Y  +590.250, Z    +0.000, E1   -36.075, E3 +394811.300}
SPL {X  -162.820, Y  +594.470, Z    +0.000, E1   -36.080, E3 +394823.531}
SPL {X  -162.820, Y  +598.788, Z    +0.000, E1   -36.102, E3 +394835.552}
SPL {X  -162.820, Y  +602.243, Z    +0.000, E1   -36.085, E3 +394845.619}
SPL {X  -162.820, Y  +605.848, Z    +0.000, E1   -36.070, E3 +394855.940}
SPL {X  -162.820, Y  +609.375, Z    +0.000, E1   -36.084, E3 +394865.991}
SPL {X  -162.820, Y  +612.959, Z    +0.000, E1   -36.034, E3 +394876.511}
SPL {X  -162.820, Y  +616.897, Z    +0.000, E1   -36.061, E3 +394887.659}
SPL {X  -162.820, Y  +621.516, Z    +0.000, E1   -36.072, E3 +394900.857}
SPL {X  -162.820, Y  +626.243, Z    +0.000, E1   -36.105, E3 +394914.100}
SPL {X  -162.820, Y  +630.571, Z    +0.000, E1   -36.057, E3 +394926.802}
SPL {X  -162.820, Y  +634.189, Z    +0.000, E1   -36.065, E3 +394936.996}
SPL {X  -162.820, Y  +638.473, Z    +0.000, E1   -36.098, E3 +394949.233}
SPL {X  -162.820, Y  +642.832, Z    +0.000, E1   -36.091, E3 +394961.559}
SPL {X  -162.820, Y  +646.320, Z    +0.000, E1   -36.078, E3 +394971.666}
SPL {X  -162.820, Y  +649.997, Z    +0.000, E1   -36.000, E3 +394982.637}
SPL {X  -162.820, Y  +655.571, Z    +0.000, E1   -36.141, E3 +394997.971}
SPL {X  -162.820, Y  +661.560, Z    +0.000, E1   -36.068, E3 +395015.398}
SPL {X  -162.820, Y  +666.386, Z    +0.000, E1   -36.048, E3 +395029.283}
SPL {X  -162.820, Y  +671.104, Z    +0.000, E1   -36.061, E3 +395042.702}
SPL {X  -162.787, Y  +676.764, Z    +0.000, E1   -36.126, E3 +395058.602}
SPL {X  -162.633, Y  +681.311, Z    +0.000, E1   -35.984, E3 +395072.290}
SPL {X  -162.367, Y  +685.641, Z    +0.000, E1   -36.000, E3 +395084.698}
SPL {X  -161.948, Y  +690.331, Z    +0.000, E1   -35.960, E3 +395098.293}
SPL {X  -161.544, Y  +693.846, Z    +0.000, E1   -35.908, E3 +395108.568}
SPL {X  -160.925, Y  +698.267, Z    +0.000, E1   -35.816, E3 +395122.001}
SPL {X  -160.151, Y  +702.861, Z    +0.000, E1   -35.643, E3 +395135.971}
SPL {X  -159.317, Y  +707.091, Z    +0.000, E1   -35.482, E3 +395149.174}
SPL {X  -158.510, Y  +710.714, Z    +0.000, E1   -35.230, E3 +395160.885}
SPL {X  -155.037, Y  +723.239, Z    +0.000, E1   -39.382, E3 +395169.981}
SPL {X  -152.141, Y  +731.494, Z    +0.000, E1   -35.181, E3 +395228.787}
ENDSPLINE

SPLINE
SPL {X  -160.133, Y  +702.956, Z    +0.000, E1   -19.806, E3 +395272.325}
SPL {X  -161.979, Y  +690.023, Z    +0.000, E1   -12.991, E3 +395275.242}
SPL {X  -162.641, Y  +681.139, Z    +0.000, E1    -7.893, E3 +395277.334}
SPL {X  -162.820, Y  +673.062, Z    +0.000, E1    -2.992, E3 +395276.301}
SPL {X  -162.820, Y  +666.731, Z    +0.000, E1    +1.545, E3 +395277.931}
SPL {X  -162.820, Y  +662.868, Z    +0.000, E1    +4.743, E3 +395278.598}
SPL {X  -162.820, Y  +657.781, Z    +0.000, E1    +9.391, E3 +395275.805}
SPL {X  -162.820, Y  +648.706, Z    +0.000, E1   +17.761, E3 +395277.556}
SPL {X  -162.820, Y  +635.926, Z    +0.000, E1   +28.192, E3 +395282.384}
SPL {X  -162.820, Y  +621.673, Z    +0.000, E1   +34.265, E3 +395298.741}
SPL {X  -162.820, Y  +609.002, Z    +0.000, E1   +38.458, E3 +395311.963}
SPL {X  -162.820, Y  +596.392, Z    +0.000, E1   +37.895, E3 +395345.432}
ENDSPLINE

SPLINE
SPL {X  -162.820, Y  +599.924, Z    +0.000, E1   +33.992, E3 +395359.806}
ENDSPLINE

SPLINE
SPL {X  -162.820, Y  +595.170, Z    +0.000, E1   +33.784, E3 +395375.854}
SPL {X  -162.820, Y  +589.785, Z    +0.000, E1   +33.904, E3 +395391.851}
SPL {X  -162.820, Y  +584.646, Z    +0.000, E1   +33.882, E3 +395407.920}
SPL {X  -162.820, Y  +579.919, Z    +0.000, E1   +33.857, E3 +395422.708}
SPL {X  -162.820, Y  +574.615, Z    +0.000, E1   +33.920, E3 +395438.882}
SPL {X  -162.820, Y  +570.335, Z    +0.000, E1   +33.821, E3 +395452.587}
SPL {X  -162.820, Y  +565.901, Z    +0.000, E1   +33.889, E3 +395466.108}
SPL {X  -162.820, Y  +562.173, Z    +0.000, E1   +33.897, E3 +395477.399}
SPL {X  -162.820, Y  +559.395, Z    +0.000, E1   +33.796, E3 +395486.766}
SPL {X  -162.820, Y  +554.453, Z    +0.000, E1   +33.841, E3 +395501.991}
SPL {X  -162.820, Y  +549.726, Z    +0.000, E1   +33.905, E3 +395516.094}
SPL {X  -162.820, Y  +545.760, Z    +0.000, E1   +33.901, E3 +395528.490}
SPL {X  -162.820, Y  +541.668, Z    +0.000, E1   +33.787, E3 +395541.890}
SPL {X  -162.820, Y  +537.061, Z    +0.000, E1   +33.897, E3 +395555.548}
SPL {X  -162.820, Y  +532.164, Z    +0.000, E1   +33.861, E3 +395571.022}
SPL {X  -162.820, Y  +528.475, Z    +0.000, E1   +33.876, E3 +395582.191}
SPL {X  -162.820, Y  +524.900, Z    +0.000, E1   +33.820, E3 +395593.850}
SPL {X  -162.820, Y  +520.532, Z    +0.000, E1   +33.805, E3 +395607.417}
SPL {X  -162.820, Y  +516.814, Z    +0.000, E1   +33.917, E3 +395618.253}
SPL {X  -162.820, Y  +512.685, Z    +0.000, E1   +33.830, E3 +395631.696}
SPL {X  -162.820, Y  +508.888, Z    +0.000, E1   +33.871, E3 +395643.111}
SPL {X  -162.820, Y  +504.570, Z    +0.000, E1   +33.876, E3 +395656.713}
SPL {X  -162.820, Y  +498.875, Z    +0.000, E1   +34.747, E3 +395668.414}
SPL {X  -162.820, Y  +481.122, Z    +0.000, E1   +41.279, E3 +395675.566}
SPL {X  -162.820, Y  +478.698, Z    +0.000, E1   +40.526, E3 +395685.915}
SPL {X  -162.820, Y  +476.364, Z    +0.000, E1   +39.976, E3 +395694.876}
SPL {X  -162.820, Y  +473.851, Z    +0.000, E1   +39.059, E3 +395707.013}
SPL {X  -162.820, Y  +470.157, Z    +0.000, E1   +38.016, E3 +395722.950}
SPL {X  -162.820, Y  +467.216, Z    +0.000, E1   +37.215, E3 +395735.712}
SPL {X  -162.820, Y  +462.598, Z    +0.000, E1   +37.325, E3 +395747.666}
SPL {X  -162.820, Y  +457.832, Z    +0.000, E1   +37.294, E3 +395760.952}
SPL {X  -162.820, Y  +452.986, Z    +0.000, E1   +37.368, E3 +395773.686}
SPL {X  -162.820, Y  +448.311, Z    +0.000, E1   +37.333, E3 +395786.706}
SPL {X  -162.820, Y  +443.351, Z    +0.000, E1   +37.335, E3 +395800.236}
SPL {X  -162.820, Y  +438.727, Z    +0.000, E1   +37.289, E3 +395813.108}
SPL {X  -162.820, Y  +434.320, Z    +0.000, E1   +37.343, E3 +395824.818}
SPL {X  -162.820, Y  +430.091, Z    +0.000, E1   +37.424, E3 +395835.818}
SPL {X  -162.820, Y  +426.177, Z    +0.000, E1   +37.250, E3 +395847.641}
SPL {X  -162.820, Y  +421.391, Z    +0.000, E1   +37.346, E3 +395860.105}
SPL {X  -162.820, Y  +416.811, Z    +0.000, E1   +37.348, E3 +395872.639}
SPL {X  -162.820, Y  +411.860, Z    +0.000, E1   +37.402, E3 +395885.791}
SPL {X  -162.820, Y  +407.726, Z    +0.000, E1   +37.291, E3 +395897.738}
SPL {X  -162.820, Y  +403.543, Z    +0.000, E1   +37.305, E3 +395909.084}
SPL {X  -162.820, Y  +399.300, Z    +0.000, E1   +37.355, E3 +395920.368}
SPL {X  -162.820, Y  +395.182, Z    +0.000, E1   +37.347, E3 +395931.657}
SPL {X  -162.820, Y  +390.797, Z    +0.000, E1   +37.358, E3 +395943.569}
SPL {X  -162.820, Y  +386.671, Z    +0.000, E1   +37.363, E3 +395954.750}
SPL {X  -162.820, Y  +382.174, Z    +0.000, E1   +37.329, E3 +395967.328}
SPL {X  -162.785, Y  +377.133, Z    +0.000, E1   +37.299, E3 +395981.257}
SPL {X  -162.576, Y  +371.586, Z    +0.000, E1   +37.322, E3 +395996.370}
SPL {X  -162.256, Y  +366.963, Z    +0.000, E1   +37.251, E3 +396009.258}
SPL {X  -161.920, Y  +363.407, Z    +0.000, E1   +37.164, E3 +396019.543}
SPL {X  -161.341, Y  +358.603, Z    +0.000, E1   +37.117, E3 +396033.024}
SPL {X  -160.616, Y  +353.801, Z    +0.000, E1   +36.942, E3 +396047.188}
SPL {X  -159.837, Y  +349.474, Z    +0.000, E1   +36.824, E3 +396059.632}
SPL {X  -159.171, Y  +346.224, Z    +0.000, E1   +36.747, E3 +396068.909}
SPL {X  -158.248, Y  +342.188, Z    +0.000, E1   +36.583, E3 +396081.071}
SPL {X  -153.520, Y  +326.260, Z    +0.000, E1   +41.363, E3 +396093.724}
SPL {X  -150.942, Y  +319.452, Z    +0.000, E1   +36.529, E3 +396150.081}
ENDSPLINE

SPLINE
SPL {X  -159.264, Y  +346.659, Z    +0.000, E1   +22.083, E3 +396190.655}
SPL {X  -161.245, Y  +357.907, Z    +0.000, E1   +16.095, E3 +396204.088}
SPL {X  -162.697, Y  +374.161, Z    +0.000, E1    +7.119, E3 +396202.077}
SPL {X  -162.820, Y  +380.878, Z    +0.000, E1    +2.854, E3 +396204.909}
SPL {X  -162.820, Y  +385.313, Z    +0.000, E1    -0.228, E3 +396204.689}
SPL {X  -162.820, Y  +389.965, Z    +0.000, E1    -3.918, E3 +396204.057}
SPL {X  -162.820, Y  +394.532, Z    +0.000, E1    -7.849, E3 +396205.605}
SPL {X  -162.820, Y  +400.765, Z    +0.000, E1   -14.108, E3 +396203.072}
SPL {X  -162.820, Y  +411.829, Z    +0.000, E1   -24.195, E3 +396205.150}
SPL {X  -162.820, Y  +434.900, Z    +0.000, E1   -34.666, E3 +396232.514}
SPL {X  -162.820, Y  +465.440, Z    +0.000, E1   -41.264, E3 +396273.822}
ENDSPLINE

SPLINE
SPL {X  -162.820, Y  +458.794, Z    +0.000, E1   -36.100, E3 +396287.445}
ENDSPLINE

SPLINE
SPL {X  -162.820, Y  +461.779, Z    +0.000, E1   -35.988, E3 +396296.641}
SPL {X  -162.820, Y  +467.031, Z    +0.000, E1   -36.178, E3 +396310.711}
SPL {X  -162.820, Y  +471.524, Z    +0.000, E1   -36.022, E3 +396324.264}
SPL {X  -162.820, Y  +475.701, Z    +0.000, E1   -36.157, E3 +396335.445}
SPL {X  -162.820, Y  +479.954, Z    +0.000, E1   -36.086, E3 +396347.986}
SPL {X  -162.820, Y  +483.976, Z    +0.000, E1   -36.049, E3 +396359.718}
SPL {X  -162.820, Y  +488.601, Z    +0.000, E1   -36.081, E3 +396372.808}
SPL {X  -162.820, Y  +493.837, Z    +0.000, E1   -36.178, E3 +396387.151}
SPL {X  -162.820, Y  +497.796, Z    +0.000, E1   -36.022, E3 +396399.336}
SPL {X  -162.820, Y  +502.146, Z    +0.000, E1   -36.123, E3 +396411.205}
SPL {X  -162.820, Y  +505.688, Z    +0.000, E1   -36.050, E3 +396421.687}
SPL {X  -162.820, Y  +509.364, Z    +0.000, E1   -36.084, E3 +396432.057}
SPL {X  -162.820, Y  +515.001, Z    +0.000, E1   -36.183, E3 +396447.695}
SPL {X  -162.820, Y  +520.482, Z    +0.000, E1   -36.096, E3 +396463.741}
SPL {X  -162.820, Y  +524.107, Z    +0.000, E1   -36.045, E3 +396474.325}
SPL {X  -162.820, Y  +527.962, Z    +0.000, E1   -36.074, E3 +396485.258}
SPL {X  -162.820, Y  +532.253, Z    +0.000, E1   -36.170, E3 +396496.847}
SPL {X  -162.820, Y  +536.031, Z    +0.000, E1   -36.058, E3 +396508.385}
SPL {X  -162.820, Y  +541.179, Z    +0.000, E1   -36.085, E3 +396523.025}
SPL {X  -162.820, Y  +546.355, Z    +0.000, E1   -36.114, E3 +396537.570}
SPL {X  -162.820, Y  +550.585, Z    +0.000, E1   -36.077, E3 +396549.839}
SPL {X  -162.820, Y  +555.903, Z    +0.000, E1   -36.136, E3 +396564.837}
SPL {X  -162.820, Y  +560.354, Z    +0.000, E1   -36.138, E3 +396577.291}
SPL {X  -162.820, Y  +562.721, Z    +0.000, E1   -36.046, E3 +396584.637}
SPL {X  -162.820, Y  +566.500, Z    +0.000, E1   -36.073, E3 +396595.369}
SPL {X  -162.820, Y  +571.734, Z    +0.000, E1   -36.094, E3 +396610.298}
SPL {X  -162.820, Y  +578.070, Z    +0.000, E1   -36.120, E3 +396628.315}
SPL {X  -162.820, Y  +582.838, Z    +0.000, E1   -36.064, E3 +396642.058}
SPL {X  -162.820, Y  +586.693, Z    +0.000, E1   -36.086, E3 +396653.034}
SPL {X  -162.820, Y  +591.665, Z    +0.000, E1   -36.045, E3 +396667.561}
SPL {X  -162.820, Y  +597.399, Z    +0.000, E1   -36.147, E3 +396683.325}
SPL {X  -162.820, Y  +602.243, Z    +0.000, E1   -36.085, E3 +396697.471}
SPL {X  -162.820, Y  +605.848, Z    +0.000, E1   -36.070, E3 +396707.792}
SPL {X  -162.820, Y  +609.375, Z    +0.000, E1   -36.084, E3 +396717.842}
SPL {X  -162.820, Y  +612.959, Z    +0.000, E1   -36.034, E3 +396728.363}
SPL {X  -162.820, Y  +616.897, Z    +0.000, E1   -36.061, E3 +396739.510}
SPL {X  -162.820, Y  +620.590, Z    +0.000, E1   -36.079, E3 +396749.905}
SPL {X  -162.820, Y  +625.276, Z    +0.000, E1   -36.104, E3 +396763.322}
SPL {X  -162.820, Y  +630.571, Z    +0.000, E1   -36.057, E3 +396778.654}
SPL {X  -162.820, Y  +634.189, Z    +0.000, E1   -36.065, E3 +396788.848}
SPL {X  -162.820, Y  +638.473, Z    +0.000, E1   -36.098, E3 +396801.085}
SPL {X  -162.820, Y  +642.832, Z    +0.000, E1   -36.091, E3 +396813.410}
SPL {X  -162.820, Y  +646.320, Z    +0.000, E1   -36.078, E3 +396823.518}
SPL {X  -162.820, Y  +651.289, Z    +0.000, E1   -36.059, E3 +396837.974}
SPL {X  -162.820, Y  +656.677, Z    +0.000, E1   -36.110, E3 +396852.987}
SPL {X  -162.820, Y  +660.489, Z    +0.000, E1   -36.068, E3 +396864.054}
SPL {X  -162.820, Y  +665.459, Z    +0.000, E1   -36.068, E3 +396878.500}
SPL {X  -162.820, Y  +672.345, Z    +0.000, E1   -36.097, E3 +396898.075}
SPL {X  -162.761, Y  +677.889, Z    +0.000, E1   -36.122, E3 +396913.540}
SPL {X  -162.633, Y  +681.311, Z    +0.000, E1   -35.984, E3 +396924.142}
SPL {X  -162.367, Y  +685.641, Z    +0.000, E1   -36.000, E3 +396936.550}
SPL {X  -162.041, Y  +689.412, Z    +0.000, E1   -36.001, E3 +396947.169}
SPL {X  -161.667, Y  +692.839, Z    +0.000, E1   -35.918, E3 +396957.591}
SPL {X  -161.078, Y  +697.256, Z    +0.000, E1   -35.797, E3 +396970.927}
SPL {X  -160.313, Y  +701.964, Z    +0.000, E1   -35.709, E3 +396985.002}
SPL {X  -159.317, Y  +707.091, Z    +0.000, E1   -35.482, E3 +397001.026}
SPL {X  -158.510, Y  +710.714, Z    +0.000, E1   -35.230, E3 +397012.737}
SPL {X  -155.037, Y  +723.239, Z    +0.000, E1   -39.382, E3 +397021.833}
SPL {X  -152.141, Y  +731.494, Z    +0.000, E1   -35.181, E3 +397080.639}
ENDSPLINE

SPLINE
SPL {X  -160.133, Y  +702.956, Z    +0.000, E1   -19.806, E3 +397124.177}
SPL {X  -161.979, Y  +690.023, Z    +0.000, E1   -12.991, E3 +397127.094}
SPL {X  -162.641, Y  +681.139, Z    +0.000, E1    -7.893, E3 +397129.186}
SPL {X  -162.820, Y  +673.062, Z    +0.000, E1    -2.992, E3 +397128.153}
SPL {X  -162.820, Y  +665.516, Z    +0.000, E1    +2.410, E3 +397129.993}
SPL {X  -162.820, Y  +657.781, Z    +0.000, E1    +9.391, E3 +397127.657}
SPL {X  -162.820, Y  +648.706, Z    +0.000, E1   +17.761, E3 +397129.408}
SPL {X  -162.820, Y  +629.267, Z    +0.000, E1   +31.872, E3 +397139.614}
SPL {X  -162.820, Y  +620.680, Z    +0.000, E1   +34.107, E3 +397153.664}
SPL {X  -162.820, Y  +601.185, Z    +0.000, E1   +39.430, E3 +397177.171}
SPL {X  -162.820, Y  +599.927, Z    +0.000, E1   +35.241, E3 +397203.749}
SPL {X  -162.820, Y  +597.570, Z    +0.000, E1   +33.919, E3 +397219.479}
SPL {X  -162.820, Y  +592.692, Z    +0.000, E1   +33.779, E3 +397235.371}
SPL {X  -162.820, Y  +588.795, Z    +0.000, E1   +33.876, E3 +397246.808}
SPL {X  -162.820, Y  +585.519, Z    +0.000, E1   +33.888, E3 +397256.892}
SPL {X  -162.820, Y  +582.066, Z    +0.000, E1   +33.857, E3 +397267.827}
SPL {X  -162.820, Y  +577.919, Z    +0.000, E1   +33.841, E3 +397280.880}
SPL {X  -162.820, Y  +573.566, Z    +0.000, E1   +33.899, E3 +397293.955}
SPL {X  -162.820, Y  +569.298, Z    +0.000, E1   +33.851, E3 +397307.596}
SPL {X  -162.820, Y  +563.983, Z    +0.000, E1   +33.916, E3 +397323.737}
SPL {X  -162.820, Y  +559.395, Z    +0.000, E1   +33.796, E3 +397338.618}
SPL {X  -162.820, Y  +554.453, Z    +0.000, E1   +33.841, E3 +397353.843}
SPL {X  -162.820, Y  +549.726, Z    +0.000, E1   +33.905, E3 +397367.946}
SPL {X  -162.820, Y  +545.760, Z    +0.000, E1   +33.901, E3 +397380.342}
SPL {X  -162.820, Y  +541.668, Z    +0.000, E1   +33.787, E3 +397393.742}
SPL {X  -162.820, Y  +537.061, Z    +0.000, E1   +33.897, E3 +397407.400}
SPL {X  -162.820, Y  +532.164, Z    +0.000, E1   +33.861, E3 +397422.874}
SPL {X  -162.820, Y  +528.475, Z    +0.000, E1   +33.876, E3 +397434.043}
SPL {X  -162.820, Y  +524.900, Z    +0.000, E1   +33.820, E3 +397445.702}
SPL {X  -162.820, Y  +520.532, Z    +0.000, E1   +33.805, E3 +397459.269}
SPL {X  -162.820, Y  +516.814, Z    +0.000, E1   +33.917, E3 +397470.105}
SPL {X  -162.820, Y  +512.685, Z    +0.000, E1   +33.830, E3 +397483.548}
SPL {X  -162.820, Y  +508.888, Z    +0.000, E1   +33.871, E3 +397494.963}
SPL {X  -162.820, Y  +505.651, Z    +0.000, E1   +33.839, E3 +397505.280}
SPL {X  -162.820, Y  +500.931, Z    +0.000, E1   +34.256, E3 +397517.153}
SPL {X  -162.820, Y  +481.122, Z    +0.000, E1   +41.279, E3 +397527.418}
SPL {X  -162.820, Y  +477.698, Z    +0.000, E1   +40.353, E3 +397541.474}
SPL {X  -162.820, Y  +474.538, Z    +0.000, E1   +39.267, E3 +397555.649}
SPL {X  -162.820, Y  +472.097, Z    +0.000, E1   +38.411, E3 +397567.193}
SPL {X  -162.820, Y  +469.308, Z    +0.000, E1   +37.839, E3 +397577.997}
SPL {X  -162.820, Y  +467.216, Z    +0.000, E1   +37.215, E3 +397587.564}
SPL {X  -162.820, Y  +462.598, Z    +0.000, E1   +37.325, E3 +397599.518}
SPL {X  -162.820, Y  +457.832, Z    +0.000, E1   +37.294, E3 +397612.804}
SPL {X  -162.820, Y  +452.986, Z    +0.000, E1   +37.368, E3 +397625.538}
SPL {X  -162.820, Y  +448.311, Z    +0.000, E1   +37.333, E3 +397638.558}
SPL {X  -162.820, Y  +443.351, Z    +0.000, E1   +37.335, E3 +397652.088}
SPL {X  -162.820, Y  +438.727, Z    +0.000, E1   +37.289, E3 +397664.960}
SPL {X  -162.820, Y  +434.320, Z    +0.000, E1   +37.343, E3 +397676.670}
SPL {X  -162.820, Y  +430.091, Z    +0.000, E1   +37.424, E3 +397687.670}
SPL {X  -162.820, Y  +426.177, Z    +0.000, E1   +37.250, E3 +397699.493}
SPL {X  -162.820, Y  +421.391, Z    +0.000, E1   +37.346, E3 +397711.957}
SPL {X  -162.820, Y  +416.811, Z    +0.000, E1   +37.348, E3 +397724.491}
SPL {X  -162.820, Y  +411.860, Z    +0.000, E1   +37.402, E3 +397737.643}
SPL {X  -162.820, Y  +407.726, Z    +0.000, E1   +37.291, E3 +397749.590}
SPL {X  -162.820, Y  +403.543, Z    +0.000, E1   +37.305, E3 +397760.936}
SPL {X  -162.820, Y  +399.300, Z    +0.000, E1   +37.355, E3 +397772.220}
SPL {X  -162.820, Y  +395.182, Z    +0.000, E1   +37.347, E3 +397783.509}
SPL {X  -162.820, Y  +390.797, Z    +0.000, E1   +37.358, E3 +397795.421}
SPL {X  -162.820, Y  +386.671, Z    +0.000, E1   +37.363, E3 +397806.602}
SPL {X  -162.820, Y  +382.174, Z    +0.000, E1   +37.329, E3 +397819.180}
SPL {X  -162.785, Y  +377.133, Z    +0.000, E1   +37.299, E3 +397833.109}
SPL {X  -162.576, Y  +371.586, Z    +0.000, E1   +37.322, E3 +397848.221}
SPL {X  -162.256, Y  +366.963, Z    +0.000, E1   +37.251, E3 +397861.110}
SPL {X  -161.920, Y  +363.407, Z    +0.000, E1   +37.164, E3 +397871.395}
SPL {X  -161.482, Y  +359.669, Z    +0.000, E1   +37.064, E3 +397882.180}
SPL {X  -160.943, Y  +355.851, Z    +0.000, E1   +37.136, E3 +397892.166}
SPL {X  -160.493, Y  +353.069, Z    +0.000, E1   +36.789, E3 +397901.818}
SPL {X  -159.837, Y  +349.474, Z    +0.000, E1   +36.824, E3 +397911.484}
SPL {X  -158.862, Y  +344.820, Z    +0.000, E1   +36.732, E3 +397924.847}
SPL {X  -157.959, Y  +341.011, Z    +0.000, E1   +36.448, E3 +397936.743}
SPL {X  -154.495, Y  +329.104, Z    +0.000, E1   +40.891, E3 +397941.626}
SPL {X  -152.543, Y  +323.569, Z    +0.000, E1   +41.772, E3 +397949.382}
SPL {X  -150.942, Y  +319.452, Z    +0.000, E1   +36.529, E3 +398001.933}
ENDSPLINE

SPLINE
SPL {X  -159.264, Y  +346.659, Z    +0.000, E1   +22.083, E3 +398042.507}
SPL {X  -161.245, Y  +357.907, Z    +0.000, E1   +16.095, E3 +398055.940}
SPL {X  -162.697, Y  +374.161, Z    +0.000, E1    +7.119, E3 +398053.929}
SPL {X  -162.820, Y  +380.878, Z    +0.000, E1    +2.854, E3 +398056.760}
SPL {X  -162.820, Y  +385.313, Z    +0.000, E1    -0.228, E3 +398056.541}
SPL {X  -162.820, Y  +389.965, Z    +0.000, E1    -3.918, E3 +398055.909}
SPL {X  -162.820, Y  +394.532, Z    +0.000, E1    -7.849, E3 +398057.457}
SPL {X  -162.820, Y  +400.765, Z    +0.000, E1   -14.108, E3 +398054.924}
SPL {X  -162.820, Y  +411.829, Z    +0.000, E1   -24.195, E3 +398057.001}
SPL {X  -162.820, Y  +434.900, Z    +0.000, E1   -34.666, E3 +398084.366}
SPL {X  -162.820, Y  +465.440, Z    +0.000, E1   -41.264, E3 +398125.674}
ENDSPLINE

SPLINE
SPL {X  -162.820, Y  +460.175, Z    +0.000, E1   -36.098, E3 +398143.473}
ENDSPLINE

SPLINE
SPL {X  -162.820, Y  +467.031, Z    +0.000, E1   -36.178, E3 +398162.563}
SPL {X  -162.820, Y  +471.524, Z    +0.000, E1   -36.022, E3 +398176.116}
SPL {X  -162.820, Y  +475.701, Z    +0.000, E1   -36.157, E3 +398187.297}
SPL {X  -162.820, Y  +479.954, Z    +0.000, E1   -36.086, E3 +398199.838}
SPL {X  -162.820, Y  +485.438, Z    +0.000, E1   -36.112, E3 +398215.556}
SPL {X  -162.820, Y  +490.843, Z    +0.000, E1   -36.087, E3 +398230.969}
SPL {X  -162.820, Y  +494.712, Z    +0.000, E1   -36.164, E3 +398241.481}
SPL {X  -162.820, Y  +497.796, Z    +0.000, E1   -36.022, E3 +398251.188}
SPL {X  -162.820, Y  +502.146, Z    +0.000, E1   -36.123, E3 +398263.057}
SPL {X  -162.820, Y  +505.688, Z    +0.000, E1   -36.050, E3 +398273.539}
SPL {X  -162.820, Y  +509.364, Z    +0.000, E1   -36.084, E3 +398283.909}
SPL {X  -162.820, Y  +515.001, Z    +0.000, E1   -36.183, E3 +398299.547}
SPL {X  -162.820, Y  +520.482, Z    +0.000, E1   -36.096, E3 +398315.593}
SPL {X  -162.820, Y  +524.107, Z    +0.000, E1   -36.045, E3 +398326.177}
SPL {X  -162.820, Y  +527.962, Z    +0.000, E1   -36.074, E3 +398337.109}
SPL {X  -162.820, Y  +532.253, Z    +0.000, E1   -36.170, E3 +398348.698}
SPL {X  -162.820, Y  +536.031, Z    +0.000, E1   -36.058, E3 +398360.236}
SPL {X  -162.820, Y  +540.096, Z    +0.000, E1   -36.040, E3 +398371.935}
SPL {X  -162.820, Y  +545.472, Z    +0.000, E1   -36.142, E3 +398386.872}
SPL {X  -162.820, Y  +550.585, Z    +0.000, E1   -36.077, E3 +398401.691}
SPL {X  -162.820, Y  +555.903, Z    +0.000, E1   -36.136, E3 +398416.689}
SPL {X  -162.820, Y  +561.684, Z    +0.000, E1   -36.118, E3 +398433.218}
SPL {X  -162.820, Y  +566.500, Z    +0.000, E1   -36.073, E3 +398447.221}
SPL {X  -162.820, Y  +571.734, Z    +0.000, E1   -36.094, E3 +398462.150}
SPL {X  -162.820, Y  +578.070, Z    +0.000, E1   -36.120, E3 +398480.167}
SPL {X  -162.820, Y  +582.838, Z    +0.000, E1   -36.064, E3 +398493.910}
SPL {X  -162.820, Y  +586.693, Z    +0.000, E1   -36.086, E3 +398504.886}
SPL {X  -162.820, Y  +591.665, Z    +0.000, E1   -36.045, E3 +398519.413}
SPL {X  -162.820, Y  +597.399, Z    +0.000, E1   -36.147, E3 +398535.177}
SPL {X  -162.820, Y  +602.243, Z    +0.000, E1   -36.085, E3 +398549.323}
SPL {X  -162.820, Y  +605.848, Z    +0.000, E1   -36.070, E3 +398559.644}
SPL {X  -162.820, Y  +609.375, Z    +0.000, E1   -36.084, E3 +398569.694}
SPL {X  -162.820, Y  +612.959, Z    +0.000, E1   -36.034, E3 +398580.215}
SPL {X  -162.820, Y  +616.897, Z    +0.000, E1   -36.061, E3 +398591.362}
SPL {X  -162.820, Y  +620.590, Z    +0.000, E1   -36.079, E3 +398601.757}
SPL {X  -162.820, Y  +625.276, Z    +0.000, E1   -36.104, E3 +398615.174}
SPL {X  -162.820, Y  +630.571, Z    +0.000, E1   -36.057, E3 +398630.506}
SPL {X  -162.820, Y  +635.505, Z    +0.000, E1   -36.079, E3 +398644.512}
SPL {X  -162.820, Y  +641.277, Z    +0.000, E1   -36.126, E3 +398660.804}
SPL {X  -162.820, Y  +646.320, Z    +0.000, E1   -36.078, E3 +398675.370}
SPL {X  -162.820, Y  +651.289, Z    +0.000, E1   -36.059, E3 +398689.826}
SPL {X  -162.820, Y  +656.677, Z    +0.000, E1   -36.110, E3 +398704.839}
SPL {X  -162.820, Y  +660.489, Z    +0.000, E1   -36.068, E3 +398715.906}
SPL {X  -162.820, Y  +665.459, Z    +0.000, E1   -36.068, E3 +398730.352}
SPL {X  -162.820, Y  +671.104, Z    +0.000, E1   -36.061, E3 +398746.406}
SPL {X  -162.787, Y  +676.764, Z    +0.000, E1   -36.126, E3 +398762.305}
SPL {X  -162.577, Y  +682.401, Z    +0.000, E1   -36.021, E3 +398779.008}
SPL {X  -162.187, Y  +687.846, Z    +0.000, E1   -36.007, E3 +398794.677}
SPL {X  -161.667, Y  +692.839, Z    +0.000, E1   -35.918, E3 +398809.443}
SPL {X  -160.925, Y  +698.267, Z    +0.000, E1   -35.816, E3 +398825.704}
SPL {X  -160.151, Y  +702.861, Z    +0.000, E1   -35.643, E3 +398839.674}
SPL {X  -159.622, Y  +705.613, Z    +0.000, E1   -35.430, E3 +398848.793}
SPL {X  -158.758, Y  +709.640, Z    +0.000, E1   -35.380, E3 +398860.800}
SPL {X  -155.037, Y  +723.239, Z    +0.000, E1   -39.382, E3 +398873.685}
SPL {X  -152.141, Y  +731.494, Z    +0.000, E1   -35.181, E3 +398932.491}
ENDSPLINE

SPLINE
SPL {X  -160.133, Y  +702.956, Z    +0.000, E1   -19.806, E3 +398976.029}
SPL {X  -161.979, Y  +690.023, Z    +0.000, E1   -12.991, E3 +398978.946}
SPL {X  -162.641, Y  +681.139, Z    +0.000, E1    -7.893, E3 +398981.038}
SPL {X  -162.820, Y  +673.062, Z    +0.000, E1    -2.992, E3 +398980.004}
SPL {X  -162.820, Y  +666.731, Z    +0.000, E1    +1.545, E3 +398981.634}
SPL {X  -162.820, Y  +660.758, Z    +0.000, E1    +6.523, E3 +398981.345}
SPL {X  -162.820, Y  +650.583, Z    +0.000, E1   +16.035, E3 +398980.317}
SPL {X  -162.820, Y  +629.267, Z    +0.000, E1   +31.872, E3 +398991.466}
SPL {X  -162.820, Y  +620.680, Z    +0.000, E1   +34.107, E3 +399005.515}
SPL {X  -162.820, Y  +609.002, Z    +0.000, E1   +38.458, E3 +399015.667}
SPL {X  -162.820, Y  +596.392, Z    +0.000, E1   +37.895, E3 +399049.136}
ENDSPLINE

SPLINE
SPL {X  -162.820, Y  +599.924, Z    +0.000, E1   +33.992, E3 +399063.509}
ENDSPLINE

SPLINE
SPL {X  -162.820, Y  +595.170, Z    +0.000, E1   +33.784, E3 +399079.558}
SPL {X  -162.820, Y  +589.785, Z    +0.000, E1   +33.904, E3 +399095.555}
SPL {X  -162.820, Y  +584.646, Z    +0.000, E1   +33.882, E3 +399111.624}
SPL {X  -162.820, Y  +579.919, Z    +0.000, E1   +33.857, E3 +399126.412}
SPL {X  -162.820, Y  +574.615, Z    +0.000, E1   +33.920, E3 +399142.586}
SPL {X  -162.820, Y  +570.335, Z    +0.000, E1   +33.821, E3 +399156.291}
SPL {X  -162.820, Y  +565.901, Z    +0.000, E1   +33.889, E3 +399169.812}
SPL {X  -162.820, Y  +560.226, Z    +0.000, E1   +33.868, E3 +399187.597}
SPL {X  -162.820, Y  +554.453, Z    +0.000, E1   +33.841, E3 +399205.695}
SPL {X  -162.820, Y  +549.726, Z    +0.000, E1   +33.905, E3 +399219.798}
SPL {X  -162.820, Y  +545.760, Z    +0.000, E1   +33.901, E3 +399232.194}
SPL {X  -162.820, Y  +541.668, Z    +0.000, E1   +33.787, E3 +399245.594}
SPL {X  -162.820, Y  +538.174, Z    +0.000, E1   +33.865, E3 +399255.883}
SPL {X  -162.820, Y  +534.943, Z    +0.000, E1   +33.919, E3 +399265.624}
SPL {X  -162.820, Y  +530.273, Z    +0.000, E1   +33.855, E3 +399280.653}
SPL {X  -162.820, Y  +524.900, Z    +0.000, E1   +33.820, E3 +399297.554}
SPL {X  -162.820, Y  +520.532, Z    +0.000, E1   +33.805, E3 +399311.121}
SPL {X  -162.820, Y  +516.814, Z    +0.000, E1   +33.917, E3 +399321.957}
SPL {X  -162.820, Y  +512.685, Z    +0.000, E1   +33.830, E3 +399335.400}
SPL {X  -162.820, Y  +508.888, Z    +0.000, E1   +33.871, E3 +399346.815}
SPL {X  -162.820, Y  +505.651, Z    +0.000, E1   +33.839, E3 +399357.132}
SPL {X  -162.820, Y  +500.931, Z    +0.000, E1   +34.256, E3 +399369.005}
SPL {X  -162.820, Y  +481.122, Z    +0.000, E1   +41.279, E3 +399379.270}
SPL {X  -162.820, Y  +478.698, Z    +0.000, E1   +40.526, E3 +399389.618}
SPL {X  -162.820, Y  +475.203, Z    +0.000, E1   +39.596, E3 +399404.078}
SPL {X  -162.820, Y  +472.097, Z    +0.000, E1   +38.411, E3 +399419.045}
SPL {X  -162.820, Y  +469.308, Z    +0.000, E1   +37.839, E3 +399429.849}
SPL {X  -162.820, Y  +467.216, Z    +0.000, E1   +37.215, E3 +399439.415}
SPL {X  -162.820, Y  +462.598, Z    +0.000, E1   +37.325, E3 +399451.370}
SPL {X  -162.820, Y  +457.832, Z    +0.000, E1   +37.294, E3 +399464.656}
SPL {X  -162.820, Y  +452.986, Z    +0.000, E1   +37.368, E3 +399477.390}
SPL {X  -162.820, Y  +448.311, Z    +0.000, E1   +37.333, E3 +399490.410}
SPL {X  -162.820, Y  +443.351, Z    +0.000, E1   +37.335, E3 +399503.940}
SPL {X  -162.820, Y  +438.727, Z    +0.000, E1   +37.289, E3 +399516.812}
SPL {X  -162.820, Y  +434.320, Z    +0.000, E1   +37.343, E3 +399528.522}
SPL {X  -162.820, Y  +430.091, Z    +0.000, E1   +37.424, E3 +399539.522}
SPL {X  -162.820, Y  +426.177, Z    +0.000, E1   +37.250, E3 +399551.345}
SPL {X  -162.820, Y  +420.241, Z    +0.000, E1   +37.355, E3 +399567.052}
SPL {X  -162.820, Y  +415.595, Z    +0.000, E1   +37.375, E3 +399579.391}
SPL {X  -162.820, Y  +411.860, Z    +0.000, E1   +37.402, E3 +399589.494}
SPL {X  -162.820, Y  +407.726, Z    +0.000, E1   +37.291, E3 +399601.442}
SPL {X  -162.820, Y  +403.543, Z    +0.000, E1   +37.305, E3 +399612.788}
SPL {X  -162.820, Y  +399.300, Z    +0.000, E1   +37.355, E3 +399624.072}
SPL {X  -162.820, Y  +395.182, Z    +0.000, E1   +37.347, E3 +399635.361}
SPL {X  -162.820, Y  +390.797, Z    +0.000, E1   +37.358, E3 +399647.273}
SPL {X  -162.820, Y  +386.671, Z    +0.000, E1   +37.363, E3 +399658.454}
SPL {X  -162.820, Y  +382.174, Z    +0.000, E1   +37.329, E3 +399671.032}
SPL {X  -162.785, Y  +377.133, Z    +0.000, E1   +37.299, E3 +399684.961}
SPL {X  -162.623, Y  +372.484, Z    +0.000, E1   +37.337, E3 +399697.400}
SPL {X  -162.331, Y  +367.894, Z    +0.000, E1   +37.251, E3 +399710.513}
SPL {X  -161.920, Y  +363.407, Z    +0.000, E1   +37.164, E3 +399723.247}
SPL {X  -161.482, Y  +359.669, Z    +0.000, E1   +37.064, E3 +399734.032}
SPL {X  -160.943, Y  +355.851, Z    +0.000, E1   +37.136, E3 +399744.018}
SPL {X  -160.493, Y  +353.069, Z    +0.000, E1   +36.789, E3 +399753.670}
SPL {X  -159.837, Y  +349.474, Z    +0.000, E1   +36.824, E3 +399763.336}
SPL {X  -159.171, Y  +346.224, Z    +0.000, E1   +36.747, E3 +399772.612}
SPL {X  -158.248, Y  +342.188, Z    +0.000, E1   +36.583, E3 +399784.775}
SPL {X  -153.520, Y  +326.260, Z    +0.000, E1   +41.363, E3 +399797.428}
SPL {X  -150.942, Y  +319.452, Z    +0.000, E1   +36.529, E3 +399853.784}
ENDSPLINE

SPLINE
SPL {X  -159.264, Y  +346.659, Z    +0.000, E1   +22.083, E3 +399894.359}
SPL {X  -161.245, Y  +357.907, Z    +0.000, E1   +16.095, E3 +399907.791}
SPL {X  -162.746, Y  +375.590, Z    +0.000, E1    +6.280, E3 +399907.380}
SPL {X  -162.820, Y  +384.478, Z    +0.000, E1    +0.434, E3 +399908.049}
SPL {X  -162.820, Y  +389.965, Z    +0.000, E1    -3.918, E3 +399907.761}
SPL {X  -162.820, Y  +394.532, Z    +0.000, E1    -7.849, E3 +399909.309}
SPL {X  -162.820, Y  +400.765, Z    +0.000, E1   -14.108, E3 +399906.776}
SPL {X  -162.820, Y  +411.829, Z    +0.000, E1   -24.195, E3 +399908.853}
SPL {X  -162.820, Y  +434.900, Z    +0.000, E1   -34.666, E3 +399936.218}
SPL {X  -162.820, Y  +465.440, Z    +0.000, E1   -41.264, E3 +399977.525}
ENDSPLINE

SPLINE
SPL {X  -162.820, Y  +460.175, Z    +0.000, E1   -36.098, E3 +399995.325}
ENDSPLINE

SPLINE
SPL {X  -162.820, Y  +465.690, Z    +0.000, E1   -36.140, E3 +400010.639}
SPL {X  -162.820, Y  +470.432, Z    +0.000, E1   -36.100, E3 +400024.522}
SPL {X  -162.820, Y  +475.701, Z    +0.000, E1   -36.157, E3 +400039.149}
SPL {X  -162.820, Y  +479.954, Z    +0.000, E1   -36.086, E3 +400051.690}
SPL {X  -162.820, Y  +483.976, Z    +0.000, E1   -36.049, E3 +400063.422}
SPL {X  -162.820, Y  +488.601, Z    +0.000, E1   -36.081, E3 +400076.512}
SPL {X  -162.820, Y  +493.837, Z    +0.000, E1   -36.178, E3 +400090.855}
SPL {X  -162.820, Y  +497.796, Z    +0.000, E1   -36.022, E3 +400103.040}
SPL {X  -162.820, Y  +502.146, Z    +0.000, E1   -36.123, E3 +400114.909}
SPL {X  -162.820, Y  +505.688, Z    +0.000, E1   -36.050, E3 +400125.390}
SPL {X  -162.820, Y  +509.364, Z    +0.000, E1   -36.084, E3 +400135.761}
SPL {X  -162.820, Y  +515.001, Z    +0.000, E1   -36.183, E3 +400151.399}
SPL {X  -162.820, Y  +520.482, Z    +0.000, E1   -36.096, E3 +400167.445}
SPL {X  -162.820, Y  +524.107, Z    +0.000, E1   -36.045, E3 +400178.028}
SPL {X  -162.820, Y  +527.962, Z    +0.000, E1   -36.074, E3 +400188.961}
SPL {X  -162.820, Y  +532.253, Z    +0.000, E1   -36.170, E3 +400200.550}
SPL {X  -162.820, Y  +536.031, Z    +0.000, E1   -36.058, E3 +400212.088}
SPL {X  -162.820, Y  +541.179, Z    +0.000, E1   -36.085, E3 +400226.729}
SPL {X  -162.820, Y  +546.355, Z    +0.000, E1   -36.114, E3 +400241.273}
SPL {X  -162.820, Y  +550.585, Z    +0.000, E1   -36.077, E3 +400253.543}
SPL {X  -162.820, Y  +555.903, Z    +0.000, E1   -36.136, E3 +400268.541}
SPL {X  -162.820, Y  +560.354, Z    +0.000, E1   -36.138, E3 +400280.995}
SPL {X  -162.820, Y  +562.721, Z    +0.000, E1   -36.046, E3 +400288.341}
SPL {X  -162.820, Y  +566.500, Z    +0.000, E1   -36.073, E3 +400299.073}
SPL {X  -162.820, Y  +570.319, Z    +0.000, E1   -36.045, E3 +400310.101}
SPL {X  -162.820, Y  +573.265, Z    +0.000, E1   -36.071, E3 +400318.337}
SPL {X  -162.820, Y  +578.070, Z    +0.000, E1   -36.120, E3 +400332.019}
SPL {X  -162.820, Y  +582.838, Z    +0.000, E1   -36.064, E3 +400345.762}
SPL {X  -162.820, Y  +586.693, Z    +0.000, E1   -36.086, E3 +400356.737}
SPL {X  -162.820, Y  +591.665, Z    +0.000, E1   -36.045, E3 +400371.265}
SPL {X  -162.820, Y  +596.059, Z    +0.000, E1   -36.124, E3 +400383.197}
SPL {X  -162.820, Y  +598.788, Z    +0.000, E1   -36.102, E3 +400391.108}
SPL {X  -162.820, Y  +602.243, Z    +0.000, E1   -36.085, E3 +400401.175}
SPL {X  -162.820, Y  +605.848, Z    +0.000, E1   -36.070, E3 +400411.496}
SPL {X  -162.820, Y  +609.375, Z    +0.000, E1   -36.084, E3 +400421.546}
SPL {X  -162.820, Y  +612.959, Z    +0.000, E1   -36.034, E3 +400432.066}
SPL {X  -162.820, Y  +616.897, Z    +0.000, E1   -36.061, E3 +400443.214}
SPL {X  -162.820, Y  +621.516, Z    +0.000, E1   -36.072, E3 +400456.413}
SPL {X  -162.820, Y  +626.243, Z    +0.000, E1   -36.105, E3 +400469.656}
SPL {X  -162.820, Y  +630.571, Z    +0.000, E1   -36.057, E3 +400482.358}
SPL {X  -162.820, Y  +635.505, Z    +0.000, E1   -36.079, E3 +400496.364}
SPL {X  -162.820, Y  +639.747, Z    +0.000, E1   -36.079, E3 +400508.390}
SPL {X  -162.820, Y  +642.832, Z    +0.000, E1   -36.091, E3 +400517.114}
SPL {X  -162.820, Y  +646.320, Z    +0.000, E1   -36.078, E3 +400527.221}
SPL {X  -162.820, Y  +651.289, Z    +0.000, E1   -36.059, E3 +400541.678}
SPL {X  -162.820, Y  +656.677, Z    +0.000, E1   -36.110, E3 +400556.691}
SPL {X  -162.820, Y  +661.560, Z    +0.000, E1   -36.068, E3 +400570.954}
SPL {X  -162.820, Y  +666.386, Z    +0.000, E1   -36.048, E3 +400584.838}
SPL {X  -162.820, Y  +672.345, Z    +0.000, E1   -36.097, E3 +400601.779}
SPL {X  -162.761, Y  +677.889, Z    +0.000, E1   -36.122, E3 +400617.243}
SPL {X  -162.577, Y  +682.401, Z    +0.000, E1   -36.021, E3 +400630.860}
SPL {X  -162.187, Y  +687.846, Z    +0.000, E1   -36.007, E3 +400646.529}
SPL {X  -161.667, Y  +692.839, Z    +0.000, E1   -35.918, E3 +400661.294}
SPL {X  -161.078, Y  +697.256, Z    +0.000, E1   -35.797, E3 +400674.631}
SPL {X  -160.313, Y  +701.964, Z    +0.000, E1   -35.709, E3 +400688.706}
SPL {X  -159.317, Y  +707.091, Z    +0.000, E1   -35.482, E3 +400704.730}
SPL {X  -158.510, Y  +710.714, Z    +0.000, E1   -35.230, E3 +400716.441}
SPL {X  -155.037, Y  +723.239, Z    +0.000, E1   -39.382, E3 +400725.537}
SPL {X  -152.141, Y  +731.494, Z    +0.000, E1   -35.181, E3 +400784.343}
ENDSPLINE

